SPLINE
SPL {X  -162.820, Y  +617.582, Z    +0.000, E1   +24.552, E3 +451834.871}
SPL {X  -162.820, Y  +614.716, Z    +0.000, E1   +24.535, E3 +451848.082}
SPL {X  -162.820, Y  +611.754, Z    +0.000, E1   +24.563, E3 +451861.370}
SPL {X  -162.820, Y  +608.970, Z    +0.000, E1   +24.542, E3 +451874.211}
SPL {X  -162.820, Y  +606.285, Z    +0.000, E1   +24.533, E3 +451886.546}
SPL {X  -162.820, Y  +603.509, Z    +0.000, E1   +24.546, E3 +451899.084}
SPL {X  -162.820, Y  +600.818, Z    +0.000, E1   +24.590, E3 +451911.006}
SPL {X  -162.820, Y  +598.053, Z    +0.000, E1   +24.547, E3 +451923.989}
SPL {X  -162.820, Y  +595.188, Z    +0.000, E1   +24.538, E3 +451937.078}
SPL {X  -162.820, Y  +592.738, Z    +0.000, E1   +24.551, E3 +451948.126}
SPL {X  -162.820, Y  +590.118, Z    +0.000, E1   +24.544, E3 +451960.185}
SPL {X  -162.820, Y  +587.204, Z    +0.000, E1   +24.592, E3 +451973.062}
SPL {X  -162.820, Y  +584.766, Z    +0.000, E1   +24.499, E3 +451984.895}
SPL {X  -162.820, Y  +581.896, Z    +0.000, E1   +24.528, E3 +451997.837}
SPL {X  -162.820, Y  +579.244, Z    +0.000, E1   +24.610, E3 +452009.181}
SPL {X  -162.820, Y  +576.848, Z    +0.000, E1   +24.543, E3 +452020.723}
SPL {X  -162.820, Y  +574.433, Z    +0.000, E1   +24.551, E3 +452031.553}
SPL {X  -162.820, Y  +572.074, Z    +0.000, E1   +24.505, E3 +452042.824}
SPL {X  -162.820, Y  +568.309, Z    +0.000, E1   +24.589, E3 +452059.451}
SPL {X  -162.820, Y  +564.977, Z    +0.000, E1   +24.571, E3 +452074.624}
SPL {X  -162.820, Y  +562.356, Z    +0.000, E1   +24.575, E3 +452086.523}
SPL {X  -162.820, Y  +558.990, Z    +0.000, E1   +24.558, E3 +452102.173}
SPL {X  -162.820, Y  +555.584, Z    +0.000, E1   +24.559, E3 +452117.541}
SPL {X  -162.820, Y  +552.867, Z    +0.000, E1   +24.583, E3 +452129.737}
SPL {X  -162.820, Y  +549.589, Z    +0.000, E1   +24.547, E3 +452145.103}
SPL {X  -162.820, Y  +545.742, Z    +0.000, E1   +24.577, E3 +452162.390}
SPL {X  -162.820, Y  +542.142, Z    +0.000, E1   +24.582, E3 +452178.743}
SPL {X  -162.820, Y  +538.903, Z    +0.000, E1   +24.519, E3 +452193.959}
SPL {X  -162.820, Y  +536.451, Z    +0.000, E1   +24.519, E3 +452205.039}
SPL {X  -162.820, Y  +534.025, Z    +0.000, E1   +24.589, E3 +452215.639}
SPL {X  -162.820, Y  +531.527, Z    +0.000, E1   +24.582, E3 +452227.024}
SPL {X  -162.820, Y  +529.165, Z    +0.000, E1   +24.521, E3 +452238.273}
SPL {X  -162.820, Y  +525.802, Z    +0.000, E1   +24.585, E3 +452253.293}
SPL {X  -162.820, Y  +521.731, Z    +0.000, E1   +24.542, E3 +452272.229}
SPL {X  -162.820, Y  +518.185, Z    +0.000, E1   +24.561, E3 +452288.101}
SPL {X  -162.820, Y  +508.728, Z    +0.000, E1   +28.484, E3 +452298.641}
SPL {X  -162.820, Y  +500.664, Z    +0.000, E1   +31.476, E3 +452307.305}
SPL {X  -162.820, Y  +499.290, Z    +0.000, E1   +30.657, E3 +452317.587}
SPL {X  -162.820, Y  +497.251, Z    +0.000, E1   +29.634, E3 +452332.063}
SPL {X  -162.820, Y  +495.647, Z    +0.000, E1   +28.606, E3 +452344.939}
SPL {X  -162.820, Y  +494.678, Z    +0.000, E1   +27.647, E3 +452355.640}
SPL {X  -162.820, Y  +493.757, Z    +0.000, E1   +26.462, E3 +452368.000}
SPL {X  -162.820, Y  +492.330, Z    +0.000, E1   +25.953, E3 +452377.754}
SPL {X  -162.820, Y  +489.800, Z    +0.000, E1   +25.653, E3 +452391.216}
SPL {X  -162.820, Y  +485.392, Z    +0.000, E1   +25.667, E3 +452410.243}
SPL {X  -162.820, Y  +482.092, Z    +0.000, E1   +25.593, E3 +452424.931}
SPL {X  -162.820, Y  +479.578, Z    +0.000, E1   +25.634, E3 +452435.574}
SPL {X  -162.820, Y  +476.226, Z    +0.000, E1   +25.672, E3 +452449.964}
SPL {X  -162.820, Y  +473.037, Z    +0.000, E1   +25.618, E3 +452464.055}
SPL {X  -162.820, Y  +469.694, Z    +0.000, E1   +25.657, E3 +452478.430}
SPL {X  -162.820, Y  +465.727, Z    +0.000, E1   +25.676, E3 +452495.473}
SPL {X  -162.820, Y  +463.001, Z    +0.000, E1   +25.614, E3 +452507.589}
SPL {X  -162.820, Y  +459.882, Z    +0.000, E1   +25.674, E3 +452520.890}
SPL {X  -162.820, Y  +456.773, Z    +0.000, E1   +25.591, E3 +452534.836}
SPL {X  -162.820, Y  +454.429, Z    +0.000, E1   +25.642, E3 +452544.604}
SPL {X  -162.820, Y  +451.204, Z    +0.000, E1   +25.672, E3 +452558.631}
SPL {X  -162.820, Y  +447.822, Z    +0.000, E1   +25.664, E3 +452573.114}
SPL {X  -162.820, Y  +445.556, Z    +0.000, E1   +25.626, E3 +452583.245}
SPL {X  -162.820, Y  +443.328, Z    +0.000, E1   +25.642, E3 +452592.759}
SPL {X  -162.820, Y  +440.857, Z    +0.000, E1   +25.614, E3 +452603.794}
SPL {X  -162.820, Y  +437.636, Z    +0.000, E1   +25.597, E3 +452617.957}
SPL {X  -162.820, Y  +434.768, Z    +0.000, E1   +25.655, E3 +452629.859}
SPL {X  -162.820, Y  +431.823, Z    +0.000, E1   +25.651, E3 +452642.858}
SPL {X  -162.820, Y  +427.740, Z    +0.000, E1   +25.667, E3 +452660.486}
SPL {X  -162.820, Y  +423.655, Z    +0.000, E1   +25.628, E3 +452678.510}
SPL {X  -162.820, Y  +419.407, Z    +0.000, E1   +25.665, E3 +452696.703}
SPL {X  -162.820, Y  +415.900, Z    +0.000, E1   +25.638, E3 +452711.972}
SPL {X  -162.820, Y  +413.088, Z    +0.000, E1   +25.644, E3 +452724.128}
SPL {X  -162.820, Y  +410.320, Z    +0.000, E1   +25.604, E3 +452736.447}
SPL {X  -162.820, Y  +407.487, Z    +0.000, E1   +25.617, E3 +452748.655}
SPL {X  -162.820, Y  +404.293, Z    +0.000, E1   +25.628, E3 +452762.564}
SPL {X  -162.820, Y  +400.835, Z    +0.000, E1   +25.694, E3 +452776.964}
SPL {X  -162.820, Y  +398.703, Z    +0.000, E1   +25.586, E3 +452786.956}
SPL {X  -162.820, Y  +396.431, Z    +0.000, E1   +25.636, E3 +452796.479}
SPL {X  -162.820, Y  +393.659, Z    +0.000, E1   +25.666, E3 +452808.329}
SPL {X  -162.820, Y  +390.679, Z    +0.000, E1   +25.624, E3 +452821.573}
SPL {X  -162.820, Y  +387.939, Z    +0.000, E1   +25.627, E3 +452833.432}
SPL {X  -162.820, Y  +384.398, Z    +0.000, E1   +25.707, E3 +452848.330}
SPL {X  -162.820, Y  +380.448, Z    +0.000, E1   +25.674, E3 +452865.694}
SPL {X  -162.785, Y  +377.106, Z    +0.000, E1   +25.598, E3 +452880.638}
SPL {X  -162.709, Y  +374.484, Z    +0.000, E1   +25.711, E3 +452891.089}
SPL {X  -162.623, Y  +372.485, Z    +0.000, E1   +25.631, E3 +452900.369}
SPL {X  -162.487, Y  +370.088, Z    +0.000, E1   +25.525, E3 +452911.623}
SPL {X  -162.243, Y  +366.801, Z    +0.000, E1   +25.618, E3 +452925.264}
SPL {X  -161.882, Y  +363.046, Z    +0.000, E1   +25.550, E3 +452942.147}
SPL {X  -161.454, Y  +359.455, Z    +0.000, E1   +25.428, E3 +452958.541}
SPL {X  -160.939, Y  +355.820, Z    +0.000, E1   +26.179, E3 +452968.424}
SPL {X  -154.424, Y  +328.890, Z    +0.000, E1   +36.591, E3 +452989.256}
ENDSPLINE

SPLINE
SPL {X  -159.701, Y  +348.785, Z    +0.000, E1   +24.361, E3 +453017.539}
SPL {X  -161.904, Y  +363.251, Z    +0.000, E1   +14.606, E3 +453047.335}
SPL {X  -162.745, Y  +375.561, Z    +0.000, E1    +7.538, E3 +453047.531}
SPL {X  -162.820, Y  +385.424, Z    +0.000, E1    +1.080, E3 +453048.425}
SPL {X  -162.820, Y  +389.940, Z    +0.000, E1    -2.281, E3 +453051.302}
SPL {X  -162.820, Y  +396.652, Z    +0.000, E1    -7.520, E3 +453050.881}
SPL {X  -162.820, Y  +406.605, Z    +0.000, E1   -16.760, E3 +453043.357}
SPL {X  -162.820, Y  +418.675, Z    +0.000, E1   -22.201, E3 +453069.606}
SPL {X  -162.820, Y  +425.113, Z    +0.000, E1   -25.243, E3 +453078.542}
SPL {X  -162.820, Y  +441.937, Z    +0.000, E1   -31.578, E3 +453100.620}
ENDSPLINE

SPLINE
SPL {X  -162.820, Y  +437.771, Z    +0.000, E1   -26.555, E3 +453119.721}
ENDSPLINE

SPLINE
SPL {X  -162.820, Y  +439.120, Z    +0.000, E1   -25.352, E3 +453134.264}
SPL {X  -162.820, Y  +441.593, Z    +0.000, E1   -25.391, E3 +453144.816}
SPL {X  -162.820, Y  +444.317, Z    +0.000, E1   -25.492, E3 +453155.997}
SPL {X  -162.820, Y  +446.544, Z    +0.000, E1   -25.427, E3 +453166.167}
SPL {X  -162.820, Y  +448.500, Z    +0.000, E1   -25.425, E3 +453174.768}
SPL {X  -162.820, Y  +451.056, Z    +0.000, E1   -25.443, E3 +453185.876}
SPL {X  -162.820, Y  +454.662, Z    +0.000, E1   -25.474, E3 +453201.620}
SPL {X  -162.820, Y  +458.079, Z    +0.000, E1   -25.369, E3 +453217.199}
SPL {X  -162.820, Y  +460.719, Z    +0.000, E1   -25.411, E3 +453228.457}
SPL {X  -162.820, Y  +463.419, Z    +0.000, E1   -25.510, E3 +453239.495}
SPL {X  -162.820, Y  +465.376, Z    +0.000, E1   -25.372, E3 +453249.083}
SPL {X  -162.820, Y  +467.440, Z    +0.000, E1   -25.427, E3 +453257.714}
SPL {X  -162.820, Y  +470.010, Z    +0.000, E1   -25.445, E3 +453268.919}
SPL {X  -162.820, Y  +473.445, Z    +0.000, E1   -25.493, E3 +453283.643}
SPL {X  -162.820, Y  +476.157, Z    +0.000, E1   -25.426, E3 +453295.858}
SPL {X  -162.820, Y  +478.461, Z    +0.000, E1   -25.410, E3 +453306.137}
SPL {X  -162.820, Y  +481.644, Z    +0.000, E1   -25.433, E3 +453320.084}
SPL {X  -162.820, Y  +486.042, Z    +0.000, E1   -25.483, E3 +453339.003}
SPL {X  -162.820, Y  +490.287, Z    +0.000, E1   -25.463, E3 +453357.721}
SPL {X  -162.820, Y  +494.454, Z    +0.000, E1   -25.465, E3 +453375.953}
SPL {X  -162.820, Y  +498.644, Z    +0.000, E1   -25.463, E3 +453394.329}
SPL {X  -162.820, Y  +502.003, Z    +0.000, E1   -25.416, E3 +453409.227}
SPL {X  -162.820, Y  +505.370, Z    +0.000, E1   -25.456, E3 +453423.803}
SPL {X  -162.820, Y  +509.412, Z    +0.000, E1   -25.458, E3 +453441.525}
SPL {X  -162.820, Y  +512.406, Z    +0.000, E1   -25.425, E3 +453454.682}
SPL {X  -162.820, Y  +515.039, Z    +0.000, E1   -25.452, E3 +453466.092}
SPL {X  -162.820, Y  +518.350, Z    +0.000, E1   -25.425, E3 +453480.842}
SPL {X  -162.820, Y  +521.486, Z    +0.000, E1   -25.382, E3 +453494.869}
SPL {X  -162.820, Y  +524.180, Z    +0.000, E1   -25.495, E3 +453505.742}
SPL {X  -162.820, Y  +527.020, Z    +0.000, E1   -25.477, E3 +453518.434}
SPL {X  -162.820, Y  +529.670, Z    +0.000, E1   -25.472, E3 +453529.892}
SPL {X  -162.820, Y  +532.006, Z    +0.000, E1   -25.455, E3 +453540.349}
SPL {X  -162.820, Y  +534.806, Z    +0.000, E1   -25.465, E3 +453552.465}
SPL {X  -162.820, Y  +537.226, Z    +0.000, E1   -25.378, E3 +453563.747}
SPL {X  -162.820, Y  +540.345, Z    +0.000, E1   -25.451, E3 +453576.928}
SPL {X  -162.820, Y  +543.279, Z    +0.000, E1   -25.419, E3 +453589.961}
SPL {X  -162.820, Y  +546.125, Z    +0.000, E1   -25.505, E3 +453601.755}
SPL {X  -162.820, Y  +549.578, Z    +0.000, E1   -25.462, E3 +453617.379}
SPL {X  -162.820, Y  +553.157, Z    +0.000, E1   -25.443, E3 +453633.043}
SPL {X  -162.820, Y  +556.150, Z    +0.000, E1   -25.445, E3 +453646.133}
SPL {X  -162.820, Y  +559.215, Z    +0.000, E1   -25.460, E3 +453659.434}
SPL {X  -162.820, Y  +562.125, Z    +0.000, E1   -25.434, E3 +453672.355}
SPL {X  -162.820, Y  +565.606, Z    +0.000, E1   -25.468, E3 +453687.484}
SPL {X  -162.820, Y  +568.974, Z    +0.000, E1   -25.453, E3 +453702.195}
SPL {X  -162.820, Y  +571.303, Z    +0.000, E1   -25.427, E3 +453712.541}
SPL {X  -162.820, Y  +574.067, Z    +0.000, E1   -25.459, E3 +453724.480}
SPL {X  -162.820, Y  +576.597, Z    +0.000, E1   -25.400, E3 +453735.951}
SPL {X  -162.820, Y  +580.038, Z    +0.000, E1   -25.473, E3 +453750.647}
SPL {X  -162.820, Y  +583.044, Z    +0.000, E1   -25.450, E3 +453763.770}
SPL {X  -162.820, Y  +585.512, Z    +0.000, E1   -25.448, E3 +453774.665}
SPL {X  -162.820, Y  +588.371, Z    +0.000, E1   -25.460, E3 +453787.051}
SPL {X  -162.820, Y  +590.476, Z    +0.000, E1   -25.398, E3 +453796.693}
SPL {X  -162.820, Y  +593.604, Z    +0.000, E1   -25.477, E3 +453809.971}
SPL {X  -162.820, Y  +596.868, Z    +0.000, E1   -25.461, E3 +453824.236}
SPL {X  -162.820, Y  +599.135, Z    +0.000, E1   -25.398, E3 +453834.605}
SPL {X  -162.820, Y  +601.296, Z    +0.000, E1   -25.399, E3 +453844.087}
SPL {X  -162.820, Y  +604.526, Z    +0.000, E1   -25.502, E3 +453857.581}
SPL {X  -162.820, Y  +607.811, Z    +0.000, E1   -25.507, E3 +453871.795}
SPL {X  -162.820, Y  +610.517, Z    +0.000, E1   -25.412, E3 +453884.358}
SPL {X  -162.820, Y  +613.762, Z    +0.000, E1   -25.472, E3 +453898.165}
SPL {X  -162.820, Y  +617.275, Z    +0.000, E1   -25.466, E3 +453913.603}
SPL {X  -162.820, Y  +619.899, Z    +0.000, E1   -25.455, E3 +453925.008}
SPL {X  -162.820, Y  +622.118, Z    +0.000, E1   -25.492, E3 +453934.475}
SPL {X  -162.820, Y  +624.430, Z    +0.000, E1   -25.475, E3 +453944.696}
SPL {X  -162.820, Y  +626.570, Z    +0.000, E1   -25.441, E3 +453954.296}
SPL {X  -162.820, Y  +628.902, Z    +0.000, E1   -25.449, E3 +453964.476}
SPL {X  -162.820, Y  +631.177, Z    +0.000, E1   -25.467, E3 +453974.308}
SPL {X  -162.820, Y  +633.994, Z    +0.000, E1   -25.503, E3 +453986.354}
SPL {X  -162.820, Y  +637.619, Z    +0.000, E1   -25.497, E3 +454002.414}
SPL {X  -162.820, Y  +640.803, Z    +0.000, E1   -25.462, E3 +454016.377}
SPL {X  -162.820, Y  +643.028, Z    +0.000, E1   -25.494, E3 +454025.886}
SPL {X  -162.820, Y  +646.519, Z    +0.000, E1   -25.551, E3 +454040.868}
SPL {X  -162.820, Y  +649.837, Z    +0.000, E1   -25.446, E3 +454055.993}
SPL {X  -162.820, Y  +652.810, Z    +0.000, E1   -25.497, E3 +454068.635}
SPL {X  -162.820, Y  +655.214, Z    +0.000, E1   -25.485, E3 +454079.138}
SPL {X  -162.820, Y  +657.616, Z    +0.000, E1   -25.511, E3 +454089.492}
SPL {X  -162.820, Y  +660.851, Z    +0.000, E1   -25.520, E3 +454103.635}
SPL {X  -162.820, Y  +663.853, Z    +0.000, E1   -25.496, E3 +454116.816}
SPL {X  -162.820, Y  +667.253, Z    +0.000, E1   -25.483, E3 +454131.989}
SPL {X  -162.820, Y  +671.102, Z    +0.000, E1   -25.514, E3 +454148.439}
SPL {X  -162.820, Y  +673.648, Z    +0.000, E1   -25.431, E3 +454160.106}
SPL {X  -162.796, Y  +676.319, Z    +0.000, E1   -25.526, E3 +454171.116}
SPL {X  -162.707, Y  +679.552, Z    +0.000, E1   -25.443, E3 +454185.990}
SPL {X  -162.545, Y  +682.952, Z    +0.000, E1   -25.510, E3 +454200.223}
SPL {X  -162.381, Y  +685.455, Z    +0.000, E1   -25.410, E3 +454211.910}
SPL {X  -162.102, Y  +688.774, Z    +0.000, E1   -25.417, E3 +454226.524}
SPL {X  -161.711, Y  +692.468, Z    +0.000, E1   -25.300, E3 +454243.497}
SPL {X  -160.732, Y  +699.494, Z    +0.000, E1   -27.462, E3 +454256.969}
SPL {X  -157.189, Y  +715.948, Z    +0.000, E1   -34.218, E3 +454269.127}
ENDSPLINE

SPLINE
SPL {X  -160.780, Y  +699.193, Z    +0.000, E1   -22.069, E3 +454301.039}
ENDSPLINE

SPLINE
SPL {X  -160.671, Y  +699.864, Z    +0.000, E1   -21.788, E3 +454308.470}
ENDSPLINE

SPLINE
SPL {X  -160.945, Y  +698.140, Z    +0.000, E1   -18.412, E3 +454346.038}
SPL {X  -162.497, Y  +683.755, Z    +0.000, E1   -10.754, E3 +454340.182}
SPL {X  -162.819, Y  +673.996, Z    +0.000, E1    -4.745, E3 +454339.783}
ENDSPLINE

SPLINE
SPL {X  -162.791, Y  +676.574, Z    +0.000, E1    -6.127, E3 +454352.471}
ENDSPLINE

SPLINE
SPL {X  -162.820, Y  +666.063, Z    +0.000, E1    +0.780, E3 +454340.564}
SPL {X  -162.820, Y  +659.251, Z    +0.000, E1    +5.716, E3 +454346.781}
SPL {X  -162.820, Y  +640.102, Z    +0.000, E1   +22.409, E3 +454342.560}
SPL {X  -162.820, Y  +633.503, Z    +0.000, E1   +21.975, E3 +454374.796}
SPL {X  -162.820, Y  +611.299, Z    +0.000, E1   +31.088, E3 +454402.909}
ENDSPLINE

SPLINE
SPL {X  -162.820, Y  +618.877, Z    +0.000, E1   +25.259, E3 +454414.403}
ENDSPLINE

SPLINE
SPL {X  -162.820, Y  +617.582, Z    +0.000, E1   +24.552, E3 +454425.780}
SPL {X  -162.820, Y  +614.716, Z    +0.000, E1   +24.535, E3 +454438.991}
SPL {X  -162.820, Y  +611.754, Z    +0.000, E1   +24.563, E3 +454452.280}
SPL {X  -162.820, Y  +608.970, Z    +0.000, E1   +24.542, E3 +454465.120}
SPL {X  -162.820, Y  +606.285, Z    +0.000, E1   +24.533, E3 +454477.455}
SPL {X  -162.820, Y  +603.509, Z    +0.000, E1   +24.546, E3 +454489.993}
SPL {X  -162.820, Y  +600.818, Z    +0.000, E1   +24.590, E3 +454501.915}
SPL {X  -162.820, Y  +598.053, Z    +0.000, E1   +24.547, E3 +454514.898}
SPL {X  -162.820, Y  +595.188, Z    +0.000, E1   +24.538, E3 +454527.987}
SPL {X  -162.820, Y  +592.738, Z    +0.000, E1   +24.551, E3 +454539.035}
SPL {X  -162.820, Y  +590.118, Z    +0.000, E1   +24.544, E3 +454551.094}
SPL {X  -162.820, Y  +587.204, Z    +0.000, E1   +24.592, E3 +454563.971}
SPL {X  -162.820, Y  +584.766, Z    +0.000, E1   +24.499, E3 +454575.804}
SPL {X  -162.820, Y  +581.896, Z    +0.000, E1   +24.528, E3 +454588.746}
SPL {X  -162.820, Y  +579.244, Z    +0.000, E1   +24.610, E3 +454600.090}
SPL {X  -162.820, Y  +576.848, Z    +0.000, E1   +24.543, E3 +454611.632}
SPL {X  -162.820, Y  +574.433, Z    +0.000, E1   +24.551, E3 +454622.462}
SPL {X  -162.820, Y  +572.074, Z    +0.000, E1   +24.505, E3 +454633.734}
SPL {X  -162.820, Y  +568.309, Z    +0.000, E1   +24.589, E3 +454650.360}
SPL {X  -162.820, Y  +564.977, Z    +0.000, E1   +24.571, E3 +454665.533}
SPL {X  -162.820, Y  +562.356, Z    +0.000, E1   +24.575, E3 +454677.432}
SPL {X  -162.820, Y  +558.990, Z    +0.000, E1   +24.558, E3 +454693.082}
SPL {X  -162.820, Y  +555.584, Z    +0.000, E1   +24.559, E3 +454708.451}
SPL {X  -162.820, Y  +552.169, Z    +0.000, E1   +24.581, E3 +454724.019}
SPL {X  -162.820, Y  +548.172, Z    +0.000, E1   +24.564, E3 +454742.367}
SPL {X  -162.820, Y  +544.025, Z    +0.000, E1   +24.611, E3 +454760.921}
SPL {X  -162.820, Y  +540.573, Z    +0.000, E1   +24.503, E3 +454777.376}
SPL {X  -162.820, Y  +537.211, Z    +0.000, E1   +24.561, E3 +454792.305}
SPL {X  -162.820, Y  +534.025, Z    +0.000, E1   +24.589, E3 +454806.548}
SPL {X  -162.820, Y  +531.527, Z    +0.000, E1   +24.582, E3 +454817.933}
SPL {X  -162.820, Y  +529.165, Z    +0.000, E1   +24.521, E3 +454829.182}
SPL {X  -162.820, Y  +526.822, Z    +0.000, E1   +24.559, E3 +454839.545}
SPL {X  -162.820, Y  +524.112, Z    +0.000, E1   +24.542, E3 +454852.163}
SPL {X  -162.820, Y  +521.048, Z    +0.000, E1   +24.515, E3 +454866.299}
SPL {X  -162.820, Y  +518.185, Z    +0.000, E1   +24.561, E3 +454879.010}
SPL {X  -162.820, Y  +508.728, Z    +0.000, E1   +28.484, E3 +454889.550}
SPL {X  -162.820, Y  +500.664, Z    +0.000, E1   +31.476, E3 +454898.214}
SPL {X  -162.820, Y  +499.290, Z    +0.000, E1   +30.657, E3 +454908.496}
SPL {X  -162.820, Y  +497.700, Z    +0.000, E1   +29.785, E3 +454920.111}
SPL {X  -162.820, Y  +495.915, Z    +0.000, E1   +28.861, E3 +454933.204}
SPL {X  -162.820, Y  +494.678, Z    +0.000, E1   +27.647, E3 +454946.549}
SPL {X  -162.820, Y  +493.757, Z    +0.000, E1   +26.462, E3 +454958.909}
SPL {X  -162.820, Y  +491.420, Z    +0.000, E1   +25.780, E3 +454974.171}
SPL {X  -162.820, Y  +487.351, Z    +0.000, E1   +25.663, E3 +454992.687}
SPL {X  -162.820, Y  +484.247, Z    +0.000, E1   +25.651, E3 +455006.013}
SPL {X  -162.820, Y  +482.092, Z    +0.000, E1   +25.593, E3 +455015.840}
SPL {X  -162.820, Y  +479.578, Z    +0.000, E1   +25.634, E3 +455026.483}
SPL {X  -162.820, Y  +477.137, Z    +0.000, E1   +25.632, E3 +455037.062}
SPL {X  -162.820, Y  +473.770, Z    +0.000, E1   +25.664, E3 +455051.608}
SPL {X  -162.820, Y  +469.694, Z    +0.000, E1   +25.657, E3 +455069.339}
SPL {X  -162.820, Y  +465.727, Z    +0.000, E1   +25.676, E3 +455086.382}
SPL {X  -162.820, Y  +463.001, Z    +0.000, E1   +25.614, E3 +455098.498}
SPL {X  -162.820, Y  +459.882, Z    +0.000, E1   +25.674, E3 +455111.799}
SPL {X  -162.820, Y  +456.773, Z    +0.000, E1   +25.591, E3 +455125.745}
SPL {X  -162.820, Y  +454.429, Z    +0.000, E1   +25.642, E3 +455135.513}
SPL {X  -162.820, Y  +451.204, Z    +0.000, E1   +25.672, E3 +455149.540}
SPL {X  -162.820, Y  +447.822, Z    +0.000, E1   +25.664, E3 +455164.023}
SPL {X  -162.820, Y  +445.556, Z    +0.000, E1   +25.626, E3 +455174.154}
SPL {X  -162.820, Y  +442.508, Z    +0.000, E1   +25.657, E3 +455187.248}
SPL {X  -162.820, Y  +439.273, Z    +0.000, E1   +25.576, E3 +455201.886}
SPL {X  -162.820, Y  +436.773, Z    +0.000, E1   +25.602, E3 +455212.451}
SPL {X  -162.820, Y  +433.761, Z    +0.000, E1   +25.681, E3 +455225.129}
SPL {X  -162.820, Y  +430.942, Z    +0.000, E1   +25.597, E3 +455237.814}
SPL {X  -162.820, Y  +428.576, Z    +0.000, E1   +25.647, E3 +455247.752}
SPL {X  -162.820, Y  +426.525, Z    +0.000, E1   +25.610, E3 +455256.860}
SPL {X  -162.820, Y  +423.655, Z    +0.000, E1   +25.628, E3 +455269.419}
SPL {X  -162.820, Y  +419.407, Z    +0.000, E1   +25.665, E3 +455287.612}
SPL {X  -162.820, Y  +415.900, Z    +0.000, E1   +25.638, E3 +455302.881}
SPL {X  -162.820, Y  +413.088, Z    +0.000, E1   +25.644, E3 +455315.037}
SPL {X  -162.820, Y  +410.320, Z    +0.000, E1   +25.604, E3 +455327.356}
SPL {X  -162.820, Y  +407.487, Z    +0.000, E1   +25.617, E3 +455339.564}
SPL {X  -162.820, Y  +405.108, Z    +0.000, E1   +25.535, E3 +455350.532}
SPL {X  -162.820, Y  +401.373, Z    +0.000, E1   +25.736, E3 +455365.368}
SPL {X  -162.820, Y  +398.703, Z    +0.000, E1   +25.586, E3 +455377.865}
SPL {X  -162.820, Y  +395.582, Z    +0.000, E1   +25.684, E3 +455390.857}
SPL {X  -162.820, Y  +391.417, Z    +0.000, E1   +25.659, E3 +455409.194}
SPL {X  -162.820, Y  +387.939, Z    +0.000, E1   +25.627, E3 +455424.341}
SPL {X  -162.820, Y  +385.565, Z    +0.000, E1   +25.686, E3 +455434.130}
SPL {X  -162.820, Y  +383.458, Z    +0.000, E1   +25.657, E3 +455443.494}
SPL {X  -162.820, Y  +381.229, Z    +0.000, E1   +25.660, E3 +455453.169}
SPL {X  -162.797, Y  +377.786, Z    +0.000, E1   +25.638, E3 +455468.459}
SPL {X  -162.663, Y  +373.346, Z    +0.000, E1   +25.707, E3 +455487.198}
SPL {X  -162.487, Y  +370.088, Z    +0.000, E1   +25.525, E3 +455502.532}
SPL {X  -162.307, Y  +367.587, Z    +0.000, E1   +25.577, E3 +455512.951}
SPL {X  -162.041, Y  +364.588, Z    +0.000, E1   +25.591, E3 +455526.028}
SPL {X  -161.695, Y  +361.389, Z    +0.000, E1   +25.445, E3 +455540.915}
SPL {X  -161.190, Y  +357.520, Z    +0.000, E1   +25.774, E3 +455555.166}
SPL {X  -155.035, Y  +330.756, Z    +0.000, E1   +37.918, E3 +455565.667}
SPL {X  -153.918, Y  +327.401, Z    +0.000, E1   +34.677, E3 +455600.968}
ENDSPLINE

SPLINE
SPL {X  -159.701, Y  +348.785, Z    +0.000, E1   +24.361, E3 +455608.449}
SPL {X  -161.904, Y  +363.251, Z    +0.000, E1   +14.606, E3 +455638.244}
SPL {X  -162.745, Y  +375.561, Z    +0.000, E1    +7.538, E3 +455638.440}
SPL {X  -162.820, Y  +385.424, Z    +0.000, E1    +1.080, E3 +455639.335}
SPL {X  -162.820, Y  +389.940, Z    +0.000, E1    -2.281, E3 +455642.211}
SPL {X  -162.820, Y  +396.652, Z    +0.000, E1    -7.520, E3 +455641.790}
SPL {X  -162.820, Y  +406.605, Z    +0.000, E1   -16.760, E3 +455634.267}
SPL {X  -162.820, Y  +420.013, Z    +0.000, E1   -22.833, E3 +455662.387}
SPL {X  -162.820, Y  +442.075, Z    +0.000, E1   -31.090, E3 +455695.173}
ENDSPLINE

SPLINE
SPL {X  -162.820, Y  +436.680, Z    +0.000, E1   -26.151, E3 +455708.478}
ENDSPLINE

SPLINE
SPL {X  -162.820, Y  +438.487, Z    +0.000, E1   -25.409, E3 +455722.117}
SPL {X  -162.820, Y  +441.593, Z    +0.000, E1   -25.391, E3 +455735.725}
SPL {X  -162.820, Y  +444.317, Z    +0.000, E1   -25.492, E3 +455746.906}
SPL {X  -162.820, Y  +447.641, Z    +0.000, E1   -25.460, E3 +455761.841}
SPL {X  -162.820, Y  +451.939, Z    +0.000, E1   -25.468, E3 +455780.662}
SPL {X  -162.820, Y  +455.480, Z    +0.000, E1   -25.454, E3 +455796.073}
SPL {X  -162.820, Y  +458.079, Z    +0.000, E1   -25.369, E3 +455808.108}
SPL {X  -162.820, Y  +460.719, Z    +0.000, E1   -25.411, E3 +455819.366}
SPL {X  -162.820, Y  +463.419, Z    +0.000, E1   -25.510, E3 +455830.404}
SPL {X  -162.820, Y  +466.458, Z    +0.000, E1   -25.433, E3 +455844.460}
SPL {X  -162.820, Y  +470.010, Z    +0.000, E1   -25.445, E3 +455859.828}
SPL {X  -162.820, Y  +472.345, Z    +0.000, E1   -25.448, E3 +455869.915}
SPL {X  -162.820, Y  +475.191, Z    +0.000, E1   -25.489, E3 +455882.277}
SPL {X  -162.820, Y  +478.461, Z    +0.000, E1   -25.410, E3 +455897.046}
SPL {X  -162.820, Y  +480.780, Z    +0.000, E1   -25.447, E3 +455906.908}
SPL {X  -162.820, Y  +483.622, Z    +0.000, E1   -25.381, E3 +455919.950}
SPL {X  -162.820, Y  +487.570, Z    +0.000, E1   -25.482, E3 +455936.588}
SPL {X  -162.820, Y  +491.017, Z    +0.000, E1   -25.445, E3 +455951.803}
SPL {X  -162.820, Y  +493.705, Z    +0.000, E1   -25.443, E3 +455963.587}
SPL {X  -162.820, Y  +497.247, Z    +0.000, E1   -25.470, E3 +455979.049}
SPL {X  -162.820, Y  +501.343, Z    +0.000, E1   -25.435, E3 +455997.248}
SPL {X  -162.820, Y  +505.370, Z    +0.000, E1   -25.456, E3 +456014.712}
SPL {X  -162.820, Y  +509.412, Z    +0.000, E1   -25.458, E3 +456032.434}
SPL {X  -162.820, Y  +512.406, Z    +0.000, E1   -25.425, E3 +456045.591}
SPL {X  -162.820, Y  +515.039, Z    +0.000, E1   -25.452, E3 +456057.001}
SPL {X  -162.820, Y  +518.350, Z    +0.000, E1   -25.425, E3 +456071.751}
SPL {X  -162.820, Y  +521.486, Z    +0.000, E1   -25.382, E3 +456085.778}
SPL {X  -162.820, Y  +524.180, Z    +0.000, E1   -25.495, E3 +456096.651}
SPL {X  -162.820, Y  +527.020, Z    +0.000, E1   -25.477, E3 +456109.343}
SPL {X  -162.820, Y  +529.670, Z    +0.000, E1   -25.472, E3 +456120.801}
SPL {X  -162.820, Y  +532.006, Z    +0.000, E1   -25.455, E3 +456131.258}
SPL {X  -162.820, Y  +534.806, Z    +0.000, E1   -25.465, E3 +456143.374}
SPL {X  -162.820, Y  +537.226, Z    +0.000, E1   -25.378, E3 +456154.656}
SPL {X  -162.820, Y  +540.345, Z    +0.000, E1   -25.451, E3 +456167.837}
SPL {X  -162.820, Y  +543.279, Z    +0.000, E1   -25.419, E3 +456180.870}
SPL {X  -162.820, Y  +546.125, Z    +0.000, E1   -25.505, E3 +456192.664}
SPL {X  -162.820, Y  +549.578, Z    +0.000, E1   -25.462, E3 +456208.289}
SPL {X  -162.820, Y  +553.157, Z    +0.000, E1   -25.443, E3 +456223.952}
SPL {X  -162.820, Y  +556.150, Z    +0.000, E1   -25.445, E3 +456237.042}
SPL {X  -162.820, Y  +559.215, Z    +0.000, E1   -25.460, E3 +456250.343}
SPL {X  -162.820, Y  +562.125, Z    +0.000, E1   -25.434, E3 +456263.264}
SPL {X  -162.820, Y  +565.606, Z    +0.000, E1   -25.468, E3 +456278.393}
SPL {X  -162.820, Y  +568.974, Z    +0.000, E1   -25.453, E3 +456293.104}
SPL {X  -162.820, Y  +571.303, Z    +0.000, E1   -25.427, E3 +456303.450}
SPL {X  -162.820, Y  +574.067, Z    +0.000, E1   -25.459, E3 +456315.389}
SPL {X  -162.820, Y  +576.597, Z    +0.000, E1   -25.400, E3 +456326.860}
SPL {X  -162.820, Y  +580.038, Z    +0.000, E1   -25.473, E3 +456341.556}
SPL {X  -162.820, Y  +583.044, Z    +0.000, E1   -25.450, E3 +456354.679}
SPL {X  -162.820, Y  +585.512, Z    +0.000, E1   -25.448, E3 +456365.575}
SPL {X  -162.820, Y  +588.371, Z    +0.000, E1   -25.460, E3 +456377.961}
SPL {X  -162.820, Y  +591.246, Z    +0.000, E1   -25.415, E3 +456390.980}
SPL {X  -162.820, Y  +594.339, Z    +0.000, E1   -25.487, E3 +456403.882}
SPL {X  -162.820, Y  +596.868, Z    +0.000, E1   -25.461, E3 +456415.145}
SPL {X  -162.820, Y  +600.326, Z    +0.000, E1   -25.438, E3 +456430.667}
SPL {X  -162.820, Y  +603.808, Z    +0.000, E1   -25.554, E3 +456444.784}
SPL {X  -162.820, Y  +607.007, Z    +0.000, E1   -25.491, E3 +456459.475}
SPL {X  -162.820, Y  +611.438, Z    +0.000, E1   -25.467, E3 +456479.065}
SPL {X  -162.820, Y  +615.388, Z    +0.000, E1   -25.455, E3 +456496.324}
SPL {X  -162.820, Y  +618.103, Z    +0.000, E1   -25.456, E3 +456508.071}
SPL {X  -162.820, Y  +621.264, Z    +0.000, E1   -25.514, E3 +456521.674}
SPL {X  -162.820, Y  +624.430, Z    +0.000, E1   -25.475, E3 +456535.605}
SPL {X  -162.820, Y  +626.570, Z    +0.000, E1   -25.441, E3 +456545.205}
SPL {X  -162.820, Y  +628.902, Z    +0.000, E1   -25.449, E3 +456555.385}
SPL {X  -162.820, Y  +631.177, Z    +0.000, E1   -25.467, E3 +456565.217}
SPL {X  -162.820, Y  +633.994, Z    +0.000, E1   -25.503, E3 +456577.263}
SPL {X  -162.820, Y  +637.619, Z    +0.000, E1   -25.497, E3 +456593.323}
SPL {X  -162.820, Y  +640.803, Z    +0.000, E1   -25.462, E3 +456607.286}
SPL {X  -162.820, Y  +643.028, Z    +0.000, E1   -25.494, E3 +456616.795}
SPL {X  -162.820, Y  +646.519, Z    +0.000, E1   -25.551, E3 +456631.777}
SPL {X  -162.820, Y  +649.837, Z    +0.000, E1   -25.446, E3 +456646.902}
SPL {X  -162.820, Y  +652.810, Z    +0.000, E1   -25.497, E3 +456659.544}
SPL {X  -162.820, Y  +655.214, Z    +0.000, E1   -25.485, E3 +456670.047}
SPL {X  -162.820, Y  +657.616, Z    +0.000, E1   -25.511, E3 +456680.401}
SPL {X  -162.820, Y  +660.851, Z    +0.000, E1   -25.520, E3 +456694.544}
SPL {X  -162.820, Y  +663.853, Z    +0.000, E1   -25.496, E3 +456707.726}
SPL {X  -162.820, Y  +667.253, Z    +0.000, E1   -25.483, E3 +456722.898}
SPL {X  -162.820, Y  +671.102, Z    +0.000, E1   -25.514, E3 +456739.348}
SPL {X  -162.820, Y  +673.648, Z    +0.000, E1   -25.431, E3 +456751.015}
SPL {X  -162.796, Y  +676.319, Z    +0.000, E1   -25.526, E3 +456762.025}
SPL {X  -162.739, Y  +678.625, Z    +0.000, E1   -25.423, E3 +456772.816}
SPL {X  -162.669, Y  +680.515, Z    +0.000, E1   -25.398, E3 +456781.270}
SPL {X  -162.545, Y  +682.952, Z    +0.000, E1   -25.510, E3 +456791.132}
SPL {X  -162.381, Y  +685.455, Z    +0.000, E1   -25.410, E3 +456802.819}
SPL {X  -162.194, Y  +687.760, Z    +0.000, E1   -25.360, E3 +456813.255}
SPL {X  -161.987, Y  +689.945, Z    +0.000, E1   -25.406, E3 +456822.407}
SPL {X  -161.711, Y  +692.468, Z    +0.000, E1   -25.300, E3 +456834.406}
SPL {X  -160.732, Y  +699.494, Z    +0.000, E1   -27.462, E3 +456847.878}
SPL {X  -157.189, Y  +715.948, Z    +0.000, E1   -34.218, E3 +456860.036}
ENDSPLINE

SPLINE
SPL {X  -157.848, Y  +713.428, Z    +0.000, E1   -28.857, E3 +456894.175}
SPL {X  -161.035, Y  +697.541, Z    +0.000, E1   -20.899, E3 +456894.694}
SPL {X  -161.689, Y  +692.657, Z    +0.000, E1   -15.656, E3 +456934.777}
SPL {X  -162.807, Y  +675.545, Z    +0.000, E1    -5.787, E3 +456930.277}
ENDSPLINE

SPLINE
SPL {X  -162.791, Y  +676.574, Z    +0.000, E1    -6.127, E3 +456943.380}
ENDSPLINE

SPLINE
SPL {X  -162.820, Y  +664.716, Z    +0.000, E1    +1.705, E3 +456932.254}
SPL {X  -162.820, Y  +658.484, Z    +0.000, E1    +6.336, E3 +456938.730}
SPL {X  -162.820, Y  +640.102, Z    +0.000, E1   +22.409, E3 +456933.469}
SPL {X  -162.820, Y  +633.503, Z    +0.000, E1   +21.975, E3 +456965.705}
SPL {X  -162.820, Y  +611.299, Z    +0.000, E1   +31.088, E3 +456993.818}
ENDSPLINE

SPLINE
SPL {X  -162.820, Y  +618.877, Z    +0.000, E1   +25.259, E3 +457005.312}
ENDSPLINE

SPLINE
SPL {X  -162.820, Y  +617.582, Z    +0.000, E1   +24.552, E3 +457016.689}
SPL {X  -162.820, Y  +614.716, Z    +0.000, E1   +24.535, E3 +457029.900}
SPL {X  -162.820, Y  +611.754, Z    +0.000, E1   +24.563, E3 +457043.189}
SPL {X  -162.820, Y  +608.970, Z    +0.000, E1   +24.542, E3 +457056.029}
SPL {X  -162.820, Y  +606.285, Z    +0.000, E1   +24.533, E3 +457068.364}
SPL {X  -162.820, Y  +603.509, Z    +0.000, E1   +24.546, E3 +457080.902}
SPL {X  -162.820, Y  +600.818, Z    +0.000, E1   +24.590, E3 +457092.824}
SPL {X  -162.820, Y  +598.053, Z    +0.000, E1   +24.547, E3 +457105.807}
SPL {X  -162.820, Y  +595.188, Z    +0.000, E1   +24.538, E3 +457118.896}
SPL {X  -162.820, Y  +592.738, Z    +0.000, E1   +24.551, E3 +457129.944}
SPL {X  -162.820, Y  +590.118, Z    +0.000, E1   +24.544, E3 +457142.003}
SPL {X  -162.820, Y  +587.204, Z    +0.000, E1   +24.592, E3 +457154.880}
SPL {X  -162.820, Y  +584.766, Z    +0.000, E1   +24.499, E3 +457166.713}
SPL {X  -162.820, Y  +581.896, Z    +0.000, E1   +24.528, E3 +457179.655}
SPL {X  -162.820, Y  +578.588, Z    +0.000, E1   +24.598, E3 +457194.207}
SPL {X  -162.820, Y  +576.196, Z    +0.000, E1   +24.519, E3 +457205.590}
SPL {X  -162.820, Y  +573.694, Z    +0.000, E1   +24.535, E3 +457217.010}
SPL {X  -162.820, Y  +570.310, Z    +0.000, E1   +24.556, E3 +457232.327}
SPL {X  -162.820, Y  +567.494, Z    +0.000, E1   +24.547, E3 +457245.112}
SPL {X  -162.820, Y  +564.977, Z    +0.000, E1   +24.571, E3 +457256.442}
SPL {X  -162.820, Y  +562.356, Z    +0.000, E1   +24.575, E3 +457268.341}
SPL {X  -162.820, Y  +558.990, Z    +0.000, E1   +24.558, E3 +457283.991}
SPL {X  -162.820, Y  +555.584, Z    +0.000, E1   +24.559, E3 +457299.360}
SPL {X  -162.820, Y  +552.169, Z    +0.000, E1   +24.581, E3 +457314.929}
SPL {X  -162.820, Y  +548.172, Z    +0.000, E1   +24.564, E3 +457333.276}
SPL {X  -162.820, Y  +544.025, Z    +0.000, E1   +24.611, E3 +457351.831}
SPL {X  -162.820, Y  +540.573, Z    +0.000, E1   +24.503, E3 +457368.285}
SPL {X  -162.820, Y  +538.106, Z    +0.000, E1   +24.553, E3 +457379.039}
SPL {X  -162.820, Y  +536.451, Z    +0.000, E1   +24.519, E3 +457386.857}
SPL {X  -162.820, Y  +534.025, Z    +0.000, E1   +24.589, E3 +457397.457}
SPL {X  -162.820, Y  +531.527, Z    +0.000, E1   +24.582, E3 +457408.843}
SPL {X  -162.820, Y  +529.165, Z    +0.000, E1   +24.521, E3 +457420.091}
SPL {X  -162.820, Y  +526.822, Z    +0.000, E1   +24.559, E3 +457430.455}
SPL {X  -162.820, Y  +524.112, Z    +0.000, E1   +24.542, E3 +457443.072}
SPL {X  -162.820, Y  +521.048, Z    +0.000, E1   +24.515, E3 +457457.209}
SPL {X  -162.820, Y  +518.185, Z    +0.000, E1   +24.561, E3 +457469.920}
SPL {X  -162.820, Y  +508.728, Z    +0.000, E1   +28.484, E3 +457480.459}
SPL {X  -162.820, Y  +500.664, Z    +0.000, E1   +31.476, E3 +457489.123}
SPL {X  -162.820, Y  +499.290, Z    +0.000, E1   +30.657, E3 +457499.405}
SPL {X  -162.820, Y  +497.251, Z    +0.000, E1   +29.634, E3 +457513.881}
SPL {X  -162.820, Y  +495.647, Z    +0.000, E1   +28.606, E3 +457526.757}
SPL {X  -162.820, Y  +494.678, Z    +0.000, E1   +27.647, E3 +457537.458}
SPL {X  -162.820, Y  +493.757, Z    +0.000, E1   +26.462, E3 +457549.818}
SPL {X  -162.820, Y  +492.330, Z    +0.000, E1   +25.953, E3 +457559.572}
SPL {X  -162.820, Y  +489.800, Z    +0.000, E1   +25.653, E3 +457573.034}
SPL {X  -162.820, Y  +485.392, Z    +0.000, E1   +25.667, E3 +457592.061}
SPL {X  -162.820, Y  +482.092, Z    +0.000, E1   +25.593, E3 +457606.749}
SPL {X  -162.820, Y  +479.578, Z    +0.000, E1   +25.634, E3 +457617.392}
SPL {X  -162.820, Y  +476.226, Z    +0.000, E1   +25.672, E3 +457631.783}
SPL {X  -162.820, Y  +473.037, Z    +0.000, E1   +25.618, E3 +457645.873}
SPL {X  -162.820, Y  +470.744, Z    +0.000, E1   +25.641, E3 +457655.614}
SPL {X  -162.820, Y  +467.745, Z    +0.000, E1   +25.668, E3 +457668.596}
SPL {X  -162.820, Y  +463.978, Z    +0.000, E1   +25.651, E3 +457685.074}
SPL {X  -162.820, Y  +459.882, Z    +0.000, E1   +25.674, E3 +457702.708}
SPL {X  -162.820, Y  +456.773, Z    +0.000, E1   +25.591, E3 +457716.654}
SPL {X  -162.820, Y  +454.429, Z    +0.000, E1   +25.642, E3 +457726.422}
SPL {X  -162.820, Y  +451.204, Z    +0.000, E1   +25.672, E3 +457740.449}
SPL {X  -162.820, Y  +447.822, Z    +0.000, E1   +25.664, E3 +457754.933}
SPL {X  -162.820, Y  +445.556, Z    +0.000, E1   +25.626, E3 +457765.063}
SPL {X  -162.820, Y  +442.508, Z    +0.000, E1   +25.657, E3 +457778.157}
SPL {X  -162.820, Y  +439.273, Z    +0.000, E1   +25.576, E3 +457792.795}
SPL {X  -162.820, Y  +436.773, Z    +0.000, E1   +25.602, E3 +457803.360}
SPL {X  -162.820, Y  +433.761, Z    +0.000, E1   +25.681, E3 +457816.038}
SPL {X  -162.820, Y  +430.942, Z    +0.000, E1   +25.597, E3 +457828.724}
SPL {X  -162.820, Y  +428.576, Z    +0.000, E1   +25.647, E3 +457838.661}
SPL {X  -162.820, Y  +425.120, Z    +0.000, E1   +25.647, E3 +457853.845}
SPL {X  -162.820, Y  +420.840, Z    +0.000, E1   +25.658, E3 +457872.352}
SPL {X  -162.820, Y  +416.590, Z    +0.000, E1   +25.659, E3 +457890.796}
SPL {X  -162.820, Y  +412.302, Z    +0.000, E1   +25.662, E3 +457909.402}
SPL {X  -162.820, Y  +408.133, Z    +0.000, E1   +25.637, E3 +457927.660}
SPL {X  -162.820, Y  +404.293, Z    +0.000, E1   +25.628, E3 +457944.382}
SPL {X  -162.820, Y  +400.835, Z    +0.000, E1   +25.694, E3 +457958.782}
SPL {X  -162.820, Y  +398.703, Z    +0.000, E1   +25.586, E3 +457968.774}
SPL {X  -162.820, Y  +395.582, Z    +0.000, E1   +25.684, E3 +457981.766}
SPL {X  -162.820, Y  +391.417, Z    +0.000, E1   +25.659, E3 +458000.104}
SPL {X  -162.820, Y  +387.939, Z    +0.000, E1   +25.627, E3 +458015.250}
SPL {X  -162.820, Y  +385.565, Z    +0.000, E1   +25.686, E3 +458025.039}
SPL {X  -162.820, Y  +383.458, Z    +0.000, E1   +25.657, E3 +458034.403}
SPL {X  -162.820, Y  +381.229, Z    +0.000, E1   +25.660, E3 +458044.078}
SPL {X  -162.797, Y  +377.786, Z    +0.000, E1   +25.638, E3 +458059.368}
SPL {X  -162.663, Y  +373.346, Z    +0.000, E1   +25.707, E3 +458078.107}
SPL {X  -162.487, Y  +370.088, Z    +0.000, E1   +25.525, E3 +458093.442}
SPL {X  -162.307, Y  +367.587, Z    +0.000, E1   +25.577, E3 +458103.860}
SPL {X  -162.041, Y  +364.588, Z    +0.000, E1   +25.591, E3 +458116.938}
SPL {X  -161.695, Y  +361.389, Z    +0.000, E1   +25.445, E3 +458131.824}
SPL {X  -161.364, Y  +358.774, Z    +0.000, E1   +25.454, E3 +458143.024}
SPL {X  -160.939, Y  +355.820, Z    +0.000, E1   +26.179, E3 +458150.242}
SPL {X  -155.035, Y  +330.756, Z    +0.000, E1   +37.918, E3 +458156.576}
SPL {X  -153.918, Y  +327.401, Z    +0.000, E1   +34.677, E3 +458191.877}
ENDSPLINE

SPLINE
SPL {X  -159.701, Y  +348.785, Z    +0.000, E1   +24.361, E3 +458199.358}
SPL {X  -161.904, Y  +363.251, Z    +0.000, E1   +14.606, E3 +458229.153}
SPL {X  -162.745, Y  +375.561, Z    +0.000, E1    +7.538, E3 +458229.349}
SPL {X  -162.820, Y  +385.424, Z    +0.000, E1    +1.080, E3 +458230.244}
SPL {X  -162.820, Y  +389.940, Z    +0.000, E1    -2.281, E3 +458233.120}
SPL {X  -162.820, Y  +396.652, Z    +0.000, E1    -7.520, E3 +458232.699}
SPL {X  -162.820, Y  +406.605, Z    +0.000, E1   -16.760, E3 +458225.176}
SPL {X  -162.820, Y  +420.013, Z    +0.000, E1   -22.833, E3 +458253.296}
SPL {X  -162.820, Y  +442.075, Z    +0.000, E1   -31.090, E3 +458286.083}
ENDSPLINE

SPLINE
SPL {X  -162.820, Y  +436.680, Z    +0.000, E1   -26.151, E3 +458299.387}
ENDSPLINE

SPLINE
SPL {X  -162.820, Y  +438.487, Z    +0.000, E1   -25.409, E3 +458313.026}
SPL {X  -162.820, Y  +441.593, Z    +0.000, E1   -25.391, E3 +458326.634}
SPL {X  -162.820, Y  +444.317, Z    +0.000, E1   -25.492, E3 +458337.815}
SPL {X  -162.820, Y  +446.544, Z    +0.000, E1   -25.427, E3 +458347.985}
SPL {X  -162.820, Y  +448.500, Z    +0.000, E1   -25.425, E3 +458356.586}
SPL {X  -162.820, Y  +451.939, Z    +0.000, E1   -25.468, E3 +458371.571}
SPL {X  -162.820, Y  +455.480, Z    +0.000, E1   -25.454, E3 +458386.982}
SPL {X  -162.820, Y  +458.079, Z    +0.000, E1   -25.369, E3 +458399.017}
SPL {X  -162.820, Y  +460.719, Z    +0.000, E1   -25.411, E3 +458410.275}
SPL {X  -162.820, Y  +463.419, Z    +0.000, E1   -25.510, E3 +458421.313}
SPL {X  -162.820, Y  +466.458, Z    +0.000, E1   -25.433, E3 +458435.369}
SPL {X  -162.820, Y  +470.010, Z    +0.000, E1   -25.445, E3 +458450.737}
SPL {X  -162.820, Y  +472.345, Z    +0.000, E1   -25.448, E3 +458460.824}
SPL {X  -162.820, Y  +475.191, Z    +0.000, E1   -25.489, E3 +458473.186}
SPL {X  -162.820, Y  +478.461, Z    +0.000, E1   -25.410, E3 +458487.955}
SPL {X  -162.820, Y  +480.780, Z    +0.000, E1   -25.447, E3 +458497.817}
SPL {X  -162.820, Y  +483.622, Z    +0.000, E1   -25.381, E3 +458510.859}
SPL {X  -162.820, Y  +487.570, Z    +0.000, E1   -25.482, E3 +458527.497}
SPL {X  -162.820, Y  +491.017, Z    +0.000, E1   -25.445, E3 +458542.712}
SPL {X  -162.820, Y  +494.454, Z    +0.000, E1   -25.465, E3 +458557.771}
SPL {X  -162.820, Y  +498.644, Z    +0.000, E1   -25.463, E3 +458576.147}
SPL {X  -162.820, Y  +502.845, Z    +0.000, E1   -25.458, E3 +458594.580}
SPL {X  -162.820, Y  +506.050, Z    +0.000, E1   -25.420, E3 +458608.720}
SPL {X  -162.820, Y  +508.346, Z    +0.000, E1   -25.444, E3 +458618.568}
SPL {X  -162.820, Y  +511.422, Z    +0.000, E1   -25.445, E3 +458632.229}
SPL {X  -162.820, Y  +515.039, Z    +0.000, E1   -25.452, E3 +458647.910}
SPL {X  -162.820, Y  +518.350, Z    +0.000, E1   -25.425, E3 +458662.660}
SPL {X  -162.820, Y  +521.486, Z    +0.000, E1   -25.382, E3 +458676.687}
SPL {X  -162.820, Y  +524.180, Z    +0.000, E1   -25.495, E3 +458687.560}
SPL {X  -162.820, Y  +527.020, Z    +0.000, E1   -25.477, E3 +458700.253}
SPL {X  -162.820, Y  +529.670, Z    +0.000, E1   -25.472, E3 +458711.710}
SPL {X  -162.820, Y  +532.006, Z    +0.000, E1   -25.455, E3 +458722.167}
SPL {X  -162.820, Y  +534.806, Z    +0.000, E1   -25.465, E3 +458734.283}
SPL {X  -162.820, Y  +537.226, Z    +0.000, E1   -25.378, E3 +458745.565}
SPL {X  -162.820, Y  +540.345, Z    +0.000, E1   -25.451, E3 +458758.746}
SPL {X  -162.820, Y  +543.279, Z    +0.000, E1   -25.419, E3 +458771.779}
SPL {X  -162.820, Y  +546.125, Z    +0.000, E1   -25.505, E3 +458783.574}
SPL {X  -162.820, Y  +548.232, Z    +0.000, E1   -25.424, E3 +458793.336}
SPL {X  -162.820, Y  +550.399, Z    +0.000, E1   -25.424, E3 +458802.887}
SPL {X  -162.820, Y  +553.157, Z    +0.000, E1   -25.443, E3 +458814.861}
SPL {X  -162.820, Y  +556.150, Z    +0.000, E1   -25.445, E3 +458827.951}
SPL {X  -162.820, Y  +559.215, Z    +0.000, E1   -25.460, E3 +458841.252}
SPL {X  -162.820, Y  +562.125, Z    +0.000, E1   -25.434, E3 +458854.173}
SPL {X  -162.820, Y  +565.606, Z    +0.000, E1   -25.468, E3 +458869.302}
SPL {X  -162.820, Y  +568.974, Z    +0.000, E1   -25.453, E3 +458884.013}
SPL {X  -162.820, Y  +571.303, Z    +0.000, E1   -25.427, E3 +458894.359}
SPL {X  -162.820, Y  +574.067, Z    +0.000, E1   -25.459, E3 +458906.298}
SPL {X  -162.820, Y  +576.597, Z    +0.000, E1   -25.400, E3 +458917.770}
SPL {X  -162.820, Y  +578.977, Z    +0.000, E1   -25.460, E3 +458927.702}
SPL {X  -162.820, Y  +581.995, Z    +0.000, E1   -25.468, E3 +458941.060}
SPL {X  -162.820, Y  +585.512, Z    +0.000, E1   -25.448, E3 +458956.484}
SPL {X  -162.820, Y  +588.371, Z    +0.000, E1   -25.460, E3 +458968.870}
SPL {X  -162.820, Y  +590.476, Z    +0.000, E1   -25.398, E3 +458978.511}
SPL {X  -162.820, Y  +593.604, Z    +0.000, E1   -25.477, E3 +458991.789}
SPL {X  -162.820, Y  +596.868, Z    +0.000, E1   -25.461, E3 +459006.054}
SPL {X  -162.820, Y  +599.135, Z    +0.000, E1   -25.398, E3 +459016.423}
SPL {X  -162.820, Y  +601.296, Z    +0.000, E1   -25.399, E3 +459025.905}
SPL {X  -162.820, Y  +603.808, Z    +0.000, E1   -25.554, E3 +459035.693}
SPL {X  -162.820, Y  +607.007, Z    +0.000, E1   -25.491, E3 +459050.384}
SPL {X  -162.820, Y  +610.517, Z    +0.000, E1   -25.412, E3 +459066.176}
SPL {X  -162.820, Y  +613.762, Z    +0.000, E1   -25.472, E3 +459079.983}
SPL {X  -162.820, Y  +617.275, Z    +0.000, E1   -25.466, E3 +459095.422}
SPL {X  -162.820, Y  +621.264, Z    +0.000, E1   -25.514, E3 +459112.583}
SPL {X  -162.820, Y  +624.430, Z    +0.000, E1   -25.475, E3 +459126.514}
SPL {X  -162.820, Y  +626.570, Z    +0.000, E1   -25.441, E3 +459136.114}
SPL {X  -162.820, Y  +628.902, Z    +0.000, E1   -25.449, E3 +459146.294}
SPL {X  -162.820, Y  +631.177, Z    +0.000, E1   -25.467, E3 +459156.126}
SPL {X  -162.820, Y  +633.994, Z    +0.000, E1   -25.503, E3 +459168.172}
SPL {X  -162.820, Y  +637.619, Z    +0.000, E1   -25.497, E3 +459184.232}
SPL {X  -162.820, Y  +640.803, Z    +0.000, E1   -25.462, E3 +459198.195}
SPL {X  -162.820, Y  +643.028, Z    +0.000, E1   -25.494, E3 +459207.704}
SPL {X  -162.820, Y  +645.694, Z    +0.000, E1   -25.540, E3 +459218.992}
SPL {X  -162.820, Y  +649.102, Z    +0.000, E1   -25.495, E3 +459234.420}
SPL {X  -162.820, Y  +652.810, Z    +0.000, E1   -25.497, E3 +459250.453}
SPL {X  -162.820, Y  +655.214, Z    +0.000, E1   -25.485, E3 +459260.956}
SPL {X  -162.820, Y  +657.616, Z    +0.000, E1   -25.511, E3 +459271.310}
SPL {X  -162.820, Y  +660.851, Z    +0.000, E1   -25.520, E3 +459285.453}
SPL {X  -162.820, Y  +663.853, Z    +0.000, E1   -25.496, E3 +459298.635}
SPL {X  -162.820, Y  +666.096, Z    +0.000, E1   -25.408, E3 +459309.102}
SPL {X  -162.820, Y  +669.195, Z    +0.000, E1   -25.525, E3 +459321.939}
SPL {X  -162.820, Y  +672.979, Z    +0.000, E1   -25.478, E3 +459338.789}
SPL {X  -162.796, Y  +676.319, Z    +0.000, E1   -25.526, E3 +459352.934}
SPL {X  -162.739, Y  +678.625, Z    +0.000, E1   -25.423, E3 +459363.725}
SPL {X  -162.669, Y  +680.515, Z    +0.000, E1   -25.398, E3 +459372.179}
SPL {X  -162.545, Y  +682.952, Z    +0.000, E1   -25.510, E3 +459382.041}
SPL {X  -162.381, Y  +685.455, Z    +0.000, E1   -25.410, E3 +459393.728}
SPL {X  -162.102, Y  +688.774, Z    +0.000, E1   -25.417, E3 +459408.342}
SPL {X  -161.711, Y  +692.468, Z    +0.000, E1   -25.300, E3 +459425.315}
SPL {X  -161.141, Y  +696.825, Z    +0.000, E1   -26.170, E3 +459437.449}
SPL {X  -157.976, Y  +712.921, Z    +0.000, E1   -33.197, E3 +459447.990}
ENDSPLINE

SPLINE
SPL {X  -160.738, Y  +699.453, Z    +0.000, E1   -21.994, E3 +459485.617}
SPL {X  -161.689, Y  +692.657, Z    +0.000, E1   -15.656, E3 +459525.686}
SPL {X  -162.807, Y  +675.545, Z    +0.000, E1    -5.787, E3 +459521.186}
ENDSPLINE

SPLINE
SPL {X  -162.791, Y  +676.574, Z    +0.000, E1    -6.127, E3 +459534.289}
ENDSPLINE

SPLINE
SPL {X  -162.820, Y  +667.935, Z    +0.000, E1    -0.509, E3 +459524.375}
SPL {X  -162.820, Y  +662.949, Z    +0.000, E1    +3.113, E3 +459522.494}
SPL {X  -162.820, Y  +659.826, Z    +0.000, E1    +5.330, E3 +459529.598}
SPL {X  -162.820, Y  +656.907, Z    +0.000, E1    +7.703, E3 +459529.688}
SPL {X  -162.820, Y  +640.102, Z    +0.000, E1   +22.409, E3 +459524.378}
SPL {X  -162.820, Y  +633.503, Z    +0.000, E1   +21.975, E3 +459556.614}
SPL {X  -162.820, Y  +611.299, Z    +0.000, E1   +31.088, E3 +459584.727}
ENDSPLINE

SPLINE
SPL {X  -162.820, Y  +618.877, Z    +0.000, E1   +25.259, E3 +459596.221}
ENDSPLINE

SPLINE
SPL {X  -162.820, Y  +617.582, Z    +0.000, E1   +24.552, E3 +459607.598}
SPL {X  -162.820, Y  +614.716, Z    +0.000, E1   +24.535, E3 +459620.810}
SPL {X  -162.820, Y  +611.754, Z    +0.000, E1   +24.563, E3 +459634.098}
SPL {X  -162.820, Y  +608.970, Z    +0.000, E1   +24.542, E3 +459646.938}
SPL {X  -162.820, Y  +606.285, Z    +0.000, E1   +24.533, E3 +459659.273}
SPL {X  -162.820, Y  +603.509, Z    +0.000, E1   +24.546, E3 +459671.811}
SPL {X  -162.820, Y  +600.818, Z    +0.000, E1   +24.590, E3 +459683.733}
SPL {X  -162.820, Y  +598.053, Z    +0.000, E1   +24.547, E3 +459696.716}
SPL {X  -162.820, Y  +595.188, Z    +0.000, E1   +24.538, E3 +459709.805}
SPL {X  -162.820, Y  +592.738, Z    +0.000, E1   +24.551, E3 +459720.853}
SPL {X  -162.820, Y  +590.118, Z    +0.000, E1   +24.544, E3 +459732.912}
SPL {X  -162.820, Y  +587.204, Z    +0.000, E1   +24.592, E3 +459745.789}
SPL {X  -162.820, Y  +584.766, Z    +0.000, E1   +24.499, E3 +459757.622}
SPL {X  -162.820, Y  +581.896, Z    +0.000, E1   +24.528, E3 +459770.564}
SPL {X  -162.820, Y  +579.244, Z    +0.000, E1   +24.610, E3 +459781.909}
SPL {X  -162.820, Y  +576.848, Z    +0.000, E1   +24.543, E3 +459793.450}
SPL {X  -162.820, Y  +573.694, Z    +0.000, E1   +24.535, E3 +459807.919}
SPL {X  -162.820, Y  +571.322, Z    +0.000, E1   +24.492, E3 +459818.953}
SPL {X  -162.820, Y  +568.309, Z    +0.000, E1   +24.589, E3 +459832.178}
SPL {X  -162.820, Y  +564.977, Z    +0.000, E1   +24.571, E3 +459847.351}
SPL {X  -162.820, Y  +562.356, Z    +0.000, E1   +24.575, E3 +459859.250}
SPL {X  -162.820, Y  +560.119, Z    +0.000, E1   +24.506, E3 +459869.938}
SPL {X  -162.820, Y  +558.093, Z    +0.000, E1   +24.537, E3 +459878.956}
SPL {X  -162.820, Y  +555.584, Z    +0.000, E1   +24.559, E3 +459890.269}
SPL {X  -162.820, Y  +552.867, Z    +0.000, E1   +24.583, E3 +459902.464}
SPL {X  -162.820, Y  +549.589, Z    +0.000, E1   +24.547, E3 +459917.830}
SPL {X  -162.820, Y  +545.742, Z    +0.000, E1   +24.577, E3 +459935.117}
SPL {X  -162.820, Y  +542.970, Z    +0.000, E1   +24.579, E3 +459947.560}
SPL {X  -162.820, Y  +540.573, Z    +0.000, E1   +24.503, E3 +459959.194}
SPL {X  -162.820, Y  +538.106, Z    +0.000, E1   +24.553, E3 +459969.948}
SPL {X  -162.820, Y  +536.451, Z    +0.000, E1   +24.519, E3 +459977.766}
SPL {X  -162.820, Y  +534.025, Z    +0.000, E1   +24.589, E3 +459988.366}
SPL {X  -162.820, Y  +531.527, Z    +0.000, E1   +24.582, E3 +459999.752}
SPL {X  -162.820, Y  +529.165, Z    +0.000, E1   +24.521, E3 +460011.000}
SPL {X  -162.820, Y  +526.822, Z    +0.000, E1   +24.559, E3 +460021.364}
SPL {X  -162.820, Y  +524.112, Z    +0.000, E1   +24.542, E3 +460033.981}
SPL {X  -162.820, Y  +521.048, Z    +0.000, E1   +24.515, E3 +460048.118}
SPL {X  -162.820, Y  +518.185, Z    +0.000, E1   +24.561, E3 +460060.829}
SPL {X  -162.820, Y  +508.728, Z    +0.000, E1   +28.484, E3 +460071.368}
SPL {X  -162.820, Y  +500.664, Z    +0.000, E1   +31.476, E3 +460080.032}
SPL {X  -162.820, Y  +499.290, Z    +0.000, E1   +30.657, E3 +460090.315}
SPL {X  -162.820, Y  +497.251, Z    +0.000, E1   +29.634, E3 +460104.790}
SPL {X  -162.820, Y  +495.647, Z    +0.000, E1   +28.606, E3 +460117.666}
SPL {X  -162.820, Y  +494.678, Z    +0.000, E1   +27.647, E3 +460128.367}
SPL {X  -162.820, Y  +493.757, Z    +0.000, E1   +26.462, E3 +460140.727}
SPL {X  -162.820, Y  +491.420, Z    +0.000, E1   +25.780, E3 +460155.989}
SPL {X  -162.820, Y  +487.351, Z    +0.000, E1   +25.663, E3 +460174.505}
SPL {X  -162.820, Y  +484.247, Z    +0.000, E1   +25.651, E3 +460187.832}
SPL {X  -162.820, Y  +482.092, Z    +0.000, E1   +25.593, E3 +460197.659}
SPL {X  -162.820, Y  +479.578, Z    +0.000, E1   +25.634, E3 +460208.301}
SPL {X  -162.820, Y  +476.226, Z    +0.000, E1   +25.672, E3 +460222.692}
SPL {X  -162.820, Y  +473.037, Z    +0.000, E1   +25.618, E3 +460236.783}
SPL {X  -162.820, Y  +469.694, Z    +0.000, E1   +25.657, E3 +460251.157}
SPL {X  -162.820, Y  +465.727, Z    +0.000, E1   +25.676, E3 +460268.200}
SPL {X  -162.820, Y  +463.001, Z    +0.000, E1   +25.614, E3 +460280.317}
SPL {X  -162.820, Y  +459.882, Z    +0.000, E1   +25.674, E3 +460293.617}
SPL {X  -162.820, Y  +456.773, Z    +0.000, E1   +25.591, E3 +460307.563}
SPL {X  -162.820, Y  +454.429, Z    +0.000, E1   +25.642, E3 +460317.331}
SPL {X  -162.820, Y  +451.204, Z    +0.000, E1   +25.672, E3 +460331.358}
SPL {X  -162.820, Y  +447.822, Z    +0.000, E1   +25.664, E3 +460345.842}
SPL {X  -162.820, Y  +445.556, Z    +0.000, E1   +25.626, E3 +460355.972}
SPL {X  -162.820, Y  +443.328, Z    +0.000, E1   +25.642, E3 +460365.487}
SPL {X  -162.820, Y  +440.857, Z    +0.000, E1   +25.614, E3 +460376.521}
SPL {X  -162.820, Y  +437.636, Z    +0.000, E1   +25.597, E3 +460390.685}
SPL {X  -162.820, Y  +434.768, Z    +0.000, E1   +25.655, E3 +460402.586}
SPL {X  -162.820, Y  +431.823, Z    +0.000, E1   +25.651, E3 +460415.585}
SPL {X  -162.820, Y  +427.740, Z    +0.000, E1   +25.667, E3 +460433.213}
SPL {X  -162.820, Y  +423.655, Z    +0.000, E1   +25.628, E3 +460451.237}
SPL {X  -162.820, Y  +419.407, Z    +0.000, E1   +25.665, E3 +460469.430}
SPL {X  -162.820, Y  +415.900, Z    +0.000, E1   +25.638, E3 +460484.699}
SPL {X  -162.820, Y  +413.088, Z    +0.000, E1   +25.644, E3 +460496.855}
SPL {X  -162.820, Y  +410.320, Z    +0.000, E1   +25.604, E3 +460509.174}
SPL {X  -162.820, Y  +407.487, Z    +0.000, E1   +25.617, E3 +460521.382}
SPL {X  -162.820, Y  +404.293, Z    +0.000, E1   +25.628, E3 +460535.291}
SPL {X  -162.820, Y  +400.835, Z    +0.000, E1   +25.694, E3 +460549.691}
SPL {X  -162.820, Y  +398.703, Z    +0.000, E1   +25.586, E3 +460559.683}
SPL {X  -162.820, Y  +395.582, Z    +0.000, E1   +25.684, E3 +460572.675}
SPL {X  -162.820, Y  +391.417, Z    +0.000, E1   +25.659, E3 +460591.013}
SPL {X  -162.820, Y  +387.939, Z    +0.000, E1   +25.627, E3 +460606.159}
SPL {X  -162.820, Y  +385.565, Z    +0.000, E1   +25.686, E3 +460615.948}
SPL {X  -162.820, Y  +383.458, Z    +0.000, E1   +25.657, E3 +460625.312}
SPL {X  -162.820, Y  +380.448, Z    +0.000, E1   +25.674, E3 +460638.421}
SPL {X  -162.785, Y  +377.106, Z    +0.000, E1   +25.598, E3 +460653.365}
SPL {X  -162.709, Y  +374.484, Z    +0.000, E1   +25.711, E3 +460663.816}
SPL {X  -162.623, Y  +372.485, Z    +0.000, E1   +25.631, E3 +460673.097}
SPL {X  -162.487, Y  +370.088, Z    +0.000, E1   +25.525, E3 +460684.351}
SPL {X  -162.243, Y  +366.801, Z    +0.000, E1   +25.618, E3 +460697.991}
SPL {X  -161.977, Y  +363.953, Z    +0.000, E1   +25.528, E3 +460710.917}
SPL {X  -161.695, Y  +361.389, Z    +0.000, E1   +25.445, E3 +460722.733}
SPL {X  -161.190, Y  +357.520, Z    +0.000, E1   +25.774, E3 +460736.984}
SPL {X  -155.035, Y  +330.756, Z    +0.000, E1   +37.918, E3 +460747.485}
SPL {X  -153.918, Y  +327.401, Z    +0.000, E1   +34.677, E3 +460782.786}
ENDSPLINE

SPLINE
SPL {X  -159.701, Y  +348.785, Z    +0.000, E1   +24.361, E3 +460790.267}
SPL {X  -162.442, Y  +369.407, Z    +0.000, E1   +11.234, E3 +460819.902}
SPL {X  -162.820, Y  +384.333, Z    +0.000, E1    +1.902, E3 +460821.108}
SPL {X  -162.820, Y  +389.940, Z    +0.000, E1    -2.281, E3 +460824.029}
SPL {X  -162.820, Y  +396.652, Z    +0.000, E1    -7.520, E3 +460823.608}
SPL {X  -162.820, Y  +406.605, Z    +0.000, E1   -16.760, E3 +460816.085}
SPL {X  -162.820, Y  +420.013, Z    +0.000, E1   -22.833, E3 +460844.206}
SPL {X  -162.820, Y  +442.075, Z    +0.000, E1   -31.090, E3 +460876.992}
ENDSPLINE

SPLINE
SPL {X  -162.820, Y  +436.680, Z    +0.000, E1   -26.151, E3 +460890.296}
ENDSPLINE

SPLINE
SPL {X  -162.820, Y  +438.487, Z    +0.000, E1   -25.409, E3 +460903.935}
SPL {X  -162.820, Y  +441.593, Z    +0.000, E1   -25.391, E3 +460917.543}
SPL {X  -162.820, Y  +444.317, Z    +0.000, E1   -25.492, E3 +460928.724}
SPL {X  -162.820, Y  +447.641, Z    +0.000, E1   -25.460, E3 +460943.660}
SPL {X  -162.820, Y  +451.056, Z    +0.000, E1   -25.443, E3 +460958.603}
SPL {X  -162.820, Y  +454.662, Z    +0.000, E1   -25.474, E3 +460974.347}
SPL {X  -162.820, Y  +458.079, Z    +0.000, E1   -25.369, E3 +460989.926}
SPL {X  -162.820, Y  +460.719, Z    +0.000, E1   -25.411, E3 +461001.184}
SPL {X  -162.820, Y  +463.419, Z    +0.000, E1   -25.510, E3 +461012.222}
SPL {X  -162.820, Y  +465.376, Z    +0.000, E1   -25.372, E3 +461021.810}
SPL {X  -162.820, Y  +467.440, Z    +0.000, E1   -25.427, E3 +461030.441}
SPL {X  -162.820, Y  +470.010, Z    +0.000, E1   -25.445, E3 +461041.646}
SPL {X  -162.820, Y  +473.445, Z    +0.000, E1   -25.493, E3 +461056.370}
SPL {X  -162.820, Y  +476.157, Z    +0.000, E1   -25.426, E3 +461068.585}
SPL {X  -162.820, Y  +478.461, Z    +0.000, E1   -25.410, E3 +461078.865}
SPL {X  -162.820, Y  +481.644, Z    +0.000, E1   -25.433, E3 +461092.811}
SPL {X  -162.820, Y  +486.042, Z    +0.000, E1   -25.483, E3 +461111.730}
SPL {X  -162.820, Y  +490.287, Z    +0.000, E1   -25.463, E3 +461130.449}
SPL {X  -162.820, Y  +494.454, Z    +0.000, E1   -25.465, E3 +461148.680}
SPL {X  -162.820, Y  +498.644, Z    +0.000, E1   -25.463, E3 +461167.056}
SPL {X  -162.820, Y  +502.003, Z    +0.000, E1   -25.416, E3 +461181.954}
SPL {X  -162.820, Y  +505.370, Z    +0.000, E1   -25.456, E3 +461196.530}
SPL {X  -162.820, Y  +509.412, Z    +0.000, E1   -25.458, E3 +461214.253}
SPL {X  -162.820, Y  +512.406, Z    +0.000, E1   -25.425, E3 +461227.409}
SPL {X  -162.820, Y  +515.039, Z    +0.000, E1   -25.452, E3 +461238.819}
SPL {X  -162.820, Y  +518.350, Z    +0.000, E1   -25.425, E3 +461253.569}
SPL {X  -162.820, Y  +521.486, Z    +0.000, E1   -25.382, E3 +461267.597}
SPL {X  -162.820, Y  +524.180, Z    +0.000, E1   -25.495, E3 +461278.469}
SPL {X  -162.820, Y  +527.020, Z    +0.000, E1   -25.477, E3 +461291.162}
SPL {X  -162.820, Y  +529.670, Z    +0.000, E1   -25.472, E3 +461302.619}
SPL {X  -162.820, Y  +532.006, Z    +0.000, E1   -25.455, E3 +461313.076}
SPL {X  -162.820, Y  +534.806, Z    +0.000, E1   -25.465, E3 +461325.193}
SPL {X  -162.820, Y  +537.226, Z    +0.000, E1   -25.378, E3 +461336.474}
SPL {X  -162.820, Y  +540.345, Z    +0.000, E1   -25.451, E3 +461349.655}
SPL {X  -162.820, Y  +543.279, Z    +0.000, E1   -25.419, E3 +461362.688}
SPL {X  -162.820, Y  +546.125, Z    +0.000, E1   -25.505, E3 +461374.483}
SPL {X  -162.820, Y  +549.578, Z    +0.000, E1   -25.462, E3 +461390.107}
SPL {X  -162.820, Y  +553.157, Z    +0.000, E1   -25.443, E3 +461405.770}
SPL {X  -162.820, Y  +556.150, Z    +0.000, E1   -25.445, E3 +461418.860}
SPL {X  -162.820, Y  +559.215, Z    +0.000, E1   -25.460, E3 +461432.162}
SPL {X  -162.820, Y  +562.125, Z    +0.000, E1   -25.434, E3 +461445.082}
SPL {X  -162.820, Y  +564.880, Z    +0.000, E1   -25.448, E3 +461457.036}
SPL {X  -162.820, Y  +568.326, Z    +0.000, E1   -25.470, E3 +461472.095}
SPL {X  -162.820, Y  +571.303, Z    +0.000, E1   -25.427, E3 +461485.268}
SPL {X  -162.820, Y  +574.067, Z    +0.000, E1   -25.459, E3 +461497.207}
SPL {X  -162.820, Y  +576.597, Z    +0.000, E1   -25.400, E3 +461508.679}
SPL {X  -162.820, Y  +578.977, Z    +0.000, E1   -25.460, E3 +461518.611}
SPL {X  -162.820, Y  +581.995, Z    +0.000, E1   -25.468, E3 +461531.969}
SPL {X  -162.820, Y  +585.512, Z    +0.000, E1   -25.448, E3 +461547.393}
SPL {X  -162.820, Y  +588.371, Z    +0.000, E1   -25.460, E3 +461559.779}
SPL {X  -162.820, Y  +591.246, Z    +0.000, E1   -25.415, E3 +461572.798}
SPL {X  -162.820, Y  +594.339, Z    +0.000, E1   -25.487, E3 +461585.700}
SPL {X  -162.820, Y  +596.868, Z    +0.000, E1   -25.461, E3 +461596.964}
SPL {X  -162.820, Y  +600.326, Z    +0.000, E1   -25.438, E3 +461612.485}
SPL {X  -162.820, Y  +604.526, Z    +0.000, E1   -25.502, E3 +461630.308}
SPL {X  -162.820, Y  +607.811, Z    +0.000, E1   -25.507, E3 +461644.523}
SPL {X  -162.820, Y  +610.517, Z    +0.000, E1   -25.412, E3 +461657.085}
SPL {X  -162.820, Y  +613.762, Z    +0.000, E1   -25.472, E3 +461670.892}
SPL {X  -162.820, Y  +617.275, Z    +0.000, E1   -25.466, E3 +461686.331}
SPL {X  -162.820, Y  +621.264, Z    +0.000, E1   -25.514, E3 +461703.492}
SPL {X  -162.820, Y  +624.430, Z    +0.000, E1   -25.475, E3 +461717.423}
SPL {X  -162.820, Y  +626.570, Z    +0.000, E1   -25.441, E3 +461727.023}
SPL {X  -162.820, Y  +628.902, Z    +0.000, E1   -25.449, E3 +461737.203}
SPL {X  -162.820, Y  +631.177, Z    +0.000, E1   -25.467, E3 +461747.035}
SPL {X  -162.820, Y  +633.994, Z    +0.000, E1   -25.503, E3 +461759.081}
SPL {X  -162.820, Y  +636.469, Z    +0.000, E1   -25.465, E3 +461770.125}
SPL {X  -162.820, Y  +638.486, Z    +0.000, E1   -25.456, E3 +461779.042}
SPL {X  -162.820, Y  +640.803, Z    +0.000, E1   -25.462, E3 +461789.104}
SPL {X  -162.820, Y  +643.028, Z    +0.000, E1   -25.494, E3 +461798.613}
SPL {X  -162.820, Y  +645.694, Z    +0.000, E1   -25.540, E3 +461809.901}
SPL {X  -162.820, Y  +649.102, Z    +0.000, E1   -25.495, E3 +461825.329}
SPL {X  -162.820, Y  +652.810, Z    +0.000, E1   -25.497, E3 +461841.362}
SPL {X  -162.820, Y  +655.214, Z    +0.000, E1   -25.485, E3 +461851.865}
SPL {X  -162.820, Y  +657.616, Z    +0.000, E1   -25.511, E3 +461862.219}
SPL {X  -162.820, Y  +660.851, Z    +0.000, E1   -25.520, E3 +461876.362}
SPL {X  -162.820, Y  +663.853, Z    +0.000, E1   -25.496, E3 +461889.544}
SPL {X  -162.820, Y  +666.096, Z    +0.000, E1   -25.408, E3 +461900.011}
SPL {X  -162.820, Y  +669.195, Z    +0.000, E1   -25.525, E3 +461912.848}
SPL {X  -162.820, Y  +672.979, Z    +0.000, E1   -25.478, E3 +461929.698}
SPL {X  -162.796, Y  +676.319, Z    +0.000, E1   -25.526, E3 +461943.843}
SPL {X  -162.739, Y  +678.625, Z    +0.000, E1   -25.423, E3 +461954.634}
SPL {X  -162.669, Y  +680.515, Z    +0.000, E1   -25.398, E3 +461963.088}
SPL {X  -162.545, Y  +682.952, Z    +0.000, E1   -25.510, E3 +461972.950}
SPL {X  -162.381, Y  +685.455, Z    +0.000, E1   -25.410, E3 +461984.637}
SPL {X  -162.194, Y  +687.760, Z    +0.000, E1   -25.360, E3 +461995.073}
SPL {X  -161.866, Y  +691.104, Z    +0.000, E1   -25.383, E3 +462009.705}
SPL {X  -161.024, Y  +697.619, Z    +0.000, E1   -26.780, E3 +462026.935}
SPL {X  -157.189, Y  +715.948, Z    +0.000, E1   -34.218, E3 +462041.854}
ENDSPLINE

SPLINE
SPL {X  -157.848, Y  +713.428, Z    +0.000, E1   -28.857, E3 +462075.994}
SPL {X  -161.035, Y  +697.541, Z    +0.000, E1   -20.899, E3 +462076.513}
SPL {X  -161.689, Y  +692.657, Z    +0.000, E1   -15.656, E3 +462116.595}
SPL {X  -162.807, Y  +675.545, Z    +0.000, E1    -5.787, E3 +462112.095}
ENDSPLINE

SPLINE
SPL {X  -162.791, Y  +676.574, Z    +0.000, E1    -6.127, E3 +462125.198}
ENDSPLINE

SPLINE
SPL {X  -162.820, Y  +664.716, Z    +0.000, E1    +1.705, E3 +462114.072}
SPL {X  -162.820, Y  +658.484, Z    +0.000, E1    +6.336, E3 +462120.548}
SPL {X  -162.820, Y  +640.102, Z    +0.000, E1   +22.409, E3 +462115.287}
SPL {X  -162.820, Y  +633.503, Z    +0.000, E1   +21.975, E3 +462147.524}
SPL {X  -162.820, Y  +611.299, Z    +0.000, E1   +31.088, E3 +462175.636}
ENDSPLINE

SPLINE
SPL {X  -162.820, Y  +618.877, Z    +0.000, E1   +25.259, E3 +462187.130}
ENDSPLINE

SPLINE
SPL {X  -162.820, Y  +617.582, Z    +0.000, E1   +24.552, E3 +462198.507}
SPL {X  -162.820, Y  +614.716, Z    +0.000, E1   +24.535, E3 +462211.719}
SPL {X  -162.820, Y  +611.754, Z    +0.000, E1   +24.563, E3 +462225.007}
SPL {X  -162.820, Y  +608.970, Z    +0.000, E1   +24.542, E3 +462237.847}
SPL {X  -162.820, Y  +606.285, Z    +0.000, E1   +24.533, E3 +462250.182}
SPL {X  -162.820, Y  +603.509, Z    +0.000, E1   +24.546, E3 +462262.720}
SPL {X  -162.820, Y  +600.818, Z    +0.000, E1   +24.590, E3 +462274.643}
SPL {X  -162.820, Y  +598.053, Z    +0.000, E1   +24.547, E3 +462287.626}
SPL {X  -162.820, Y  +595.188, Z    +0.000, E1   +24.538, E3 +462300.714}
SPL {X  -162.820, Y  +592.738, Z    +0.000, E1   +24.551, E3 +462311.762}
SPL {X  -162.820, Y  +590.118, Z    +0.000, E1   +24.544, E3 +462323.821}
SPL {X  -162.820, Y  +587.204, Z    +0.000, E1   +24.592, E3 +462336.698}
SPL {X  -162.820, Y  +584.193, Z    +0.000, E1   +24.484, E3 +462351.408}
SPL {X  -162.820, Y  +580.163, Z    +0.000, E1   +24.634, E3 +462368.643}
SPL {X  -162.820, Y  +576.848, Z    +0.000, E1   +24.543, E3 +462384.359}
SPL {X  -162.820, Y  +574.433, Z    +0.000, E1   +24.551, E3 +462395.190}
SPL {X  -162.820, Y  +572.074, Z    +0.000, E1   +24.505, E3 +462406.461}
SPL {X  -162.820, Y  +569.438, Z    +0.000, E1   +24.562, E3 +462417.920}
SPL {X  -162.820, Y  +567.494, Z    +0.000, E1   +24.547, E3 +462426.930}
SPL {X  -162.820, Y  +564.977, Z    +0.000, E1   +24.571, E3 +462438.260}
SPL {X  -162.820, Y  +562.356, Z    +0.000, E1   +24.575, E3 +462450.159}
SPL {X  -162.820, Y  +560.119, Z    +0.000, E1   +24.506, E3 +462460.848}
SPL {X  -162.820, Y  +558.093, Z    +0.000, E1   +24.537, E3 +462469.865}
SPL {X  -162.820, Y  +555.584, Z    +0.000, E1   +24.559, E3 +462481.178}
SPL {X  -162.820, Y  +552.169, Z    +0.000, E1   +24.581, E3 +462496.747}
SPL {X  -162.820, Y  +548.932, Z    +0.000, E1   +24.540, E3 +462511.647}
SPL {X  -162.820, Y  +545.742, Z    +0.000, E1   +24.577, E3 +462526.026}
SPL {X  -162.820, Y  +542.142, Z    +0.000, E1   +24.582, E3 +462542.379}
SPL {X  -162.820, Y  +538.903, Z    +0.000, E1   +24.519, E3 +462557.595}
SPL {X  -162.820, Y  +536.451, Z    +0.000, E1   +24.519, E3 +462568.675}
SPL {X  -162.820, Y  +534.025, Z    +0.000, E1   +24.589, E3 +462579.275}
SPL {X  -162.820, Y  +531.527, Z    +0.000, E1   +24.582, E3 +462590.661}
SPL {X  -162.820, Y  +529.165, Z    +0.000, E1   +24.521, E3 +462601.910}
SPL {X  -162.820, Y  +526.822, Z    +0.000, E1   +24.559, E3 +462612.273}
SPL {X  -162.820, Y  +524.112, Z    +0.000, E1   +24.542, E3 +462624.890}
SPL {X  -162.820, Y  +521.048, Z    +0.000, E1   +24.515, E3 +462639.027}
SPL {X  -162.820, Y  +518.185, Z    +0.000, E1   +24.561, E3 +462651.738}
SPL {X  -162.820, Y  +508.728, Z    +0.000, E1   +28.484, E3 +462662.278}
SPL {X  -162.820, Y  +500.664, Z    +0.000, E1   +31.476, E3 +462670.942}
SPL {X  -162.820, Y  +499.290, Z    +0.000, E1   +30.657, E3 +462681.224}
SPL {X  -162.820, Y  +497.700, Z    +0.000, E1   +29.785, E3 +462692.838}
SPL {X  -162.820, Y  +495.915, Z    +0.000, E1   +28.861, E3 +462705.931}
SPL {X  -162.820, Y  +494.678, Z    +0.000, E1   +27.647, E3 +462719.276}
SPL {X  -162.820, Y  +493.757, Z    +0.000, E1   +26.462, E3 +462731.636}
SPL {X  -162.820, Y  +491.420, Z    +0.000, E1   +25.780, E3 +462746.898}
SPL {X  -162.820, Y  +487.351, Z    +0.000, E1   +25.663, E3 +462765.414}
SPL {X  -162.820, Y  +484.247, Z    +0.000, E1   +25.651, E3 +462778.741}
SPL {X  -162.820, Y  +482.092, Z    +0.000, E1   +25.593, E3 +462788.568}
SPL {X  -162.820, Y  +479.578, Z    +0.000, E1   +25.634, E3 +462799.210}
SPL {X  -162.820, Y  +477.137, Z    +0.000, E1   +25.632, E3 +462809.790}
SPL {X  -162.820, Y  +473.770, Z    +0.000, E1   +25.664, E3 +462824.335}
SPL {X  -162.820, Y  +469.694, Z    +0.000, E1   +25.657, E3 +462842.067}
SPL {X  -162.820, Y  +465.727, Z    +0.000, E1   +25.676, E3 +462859.110}
SPL {X  -162.820, Y  +463.001, Z    +0.000, E1   +25.614, E3 +462871.226}
SPL {X  -162.820, Y  +459.882, Z    +0.000, E1   +25.674, E3 +462884.526}
SPL {X  -162.820, Y  +456.773, Z    +0.000, E1   +25.591, E3 +462898.472}
SPL {X  -162.820, Y  +454.429, Z    +0.000, E1   +25.642, E3 +462908.240}
SPL {X  -162.820, Y  +451.204, Z    +0.000, E1   +25.672, E3 +462922.267}
SPL {X  -162.820, Y  +447.822, Z    +0.000, E1   +25.664, E3 +462936.751}
SPL {X  -162.820, Y  +445.556, Z    +0.000, E1   +25.626, E3 +462946.882}
SPL {X  -162.820, Y  +443.328, Z    +0.000, E1   +25.642, E3 +462956.396}
SPL {X  -162.820, Y  +440.857, Z    +0.000, E1   +25.614, E3 +462967.430}
SPL {X  -162.820, Y  +437.636, Z    +0.000, E1   +25.597, E3 +462981.594}
SPL {X  -162.820, Y  +434.768, Z    +0.000, E1   +25.655, E3 +462993.495}
SPL {X  -162.820, Y  +431.823, Z    +0.000, E1   +25.651, E3 +463006.494}
SPL {X  -162.820, Y  +427.740, Z    +0.000, E1   +25.667, E3 +463024.122}
SPL {X  -162.820, Y  +423.655, Z    +0.000, E1   +25.628, E3 +463042.147}
SPL {X  -162.820, Y  +419.407, Z    +0.000, E1   +25.665, E3 +463060.339}
SPL {X  -162.820, Y  +415.900, Z    +0.000, E1   +25.638, E3 +463075.608}
SPL {X  -162.820, Y  +413.088, Z    +0.000, E1   +25.644, E3 +463087.764}
SPL {X  -162.820, Y  +410.320, Z    +0.000, E1   +25.604, E3 +463100.083}
SPL {X  -162.820, Y  +407.487, Z    +0.000, E1   +25.617, E3 +463112.291}
SPL {X  -162.820, Y  +405.108, Z    +0.000, E1   +25.535, E3 +463123.259}
SPL {X  -162.820, Y  +401.373, Z    +0.000, E1   +25.736, E3 +463138.095}
SPL {X  -162.820, Y  +398.703, Z    +0.000, E1   +25.586, E3 +463150.592}
SPL {X  -162.820, Y  +395.582, Z    +0.000, E1   +25.684, E3 +463163.584}
SPL {X  -162.820, Y  +391.417, Z    +0.000, E1   +25.659, E3 +463181.922}
SPL {X  -162.820, Y  +387.939, Z    +0.000, E1   +25.627, E3 +463197.069}
SPL {X  -162.820, Y  +385.565, Z    +0.000, E1   +25.686, E3 +463206.857}
SPL {X  -162.820, Y  +383.458, Z    +0.000, E1   +25.657, E3 +463216.221}
SPL {X  -162.820, Y  +381.229, Z    +0.000, E1   +25.660, E3 +463225.897}
SPL {X  -162.797, Y  +377.786, Z    +0.000, E1   +25.638, E3 +463241.186}
SPL {X  -162.663, Y  +373.346, Z    +0.000, E1   +25.707, E3 +463259.925}
SPL {X  -162.487, Y  +370.088, Z    +0.000, E1   +25.525, E3 +463275.260}
SPL {X  -162.307, Y  +367.587, Z    +0.000, E1   +25.577, E3 +463285.678}
SPL {X  -162.041, Y  +364.588, Z    +0.000, E1   +25.591, E3 +463298.756}
SPL {X  -161.695, Y  +361.389, Z    +0.000, E1   +25.445, E3 +463313.642}
SPL {X  -161.364, Y  +358.774, Z    +0.000, E1   +25.454, E3 +463324.842}
SPL {X  -160.939, Y  +355.820, Z    +0.000, E1   +26.179, E3 +463332.060}
SPL {X  -155.035, Y  +330.756, Z    +0.000, E1   +37.918, E3 +463338.394}
SPL {X  -153.918, Y  +327.401, Z    +0.000, E1   +34.677, E3 +463373.695}
ENDSPLINE

SPLINE
SPL {X  -159.701, Y  +348.785, Z    +0.000, E1   +24.361, E3 +463381.176}
SPL {X  -162.442, Y  +369.407, Z    +0.000, E1   +11.234, E3 +463410.811}
SPL {X  -162.820, Y  +384.333, Z    +0.000, E1    +1.902, E3 +463412.017}
SPL {X  -162.820, Y  +389.940, Z    +0.000, E1    -2.281, E3 +463414.938}
SPL {X  -162.820, Y  +396.652, Z    +0.000, E1    -7.520, E3 +463414.517}
SPL {X  -162.820, Y  +409.181, Z    +0.000, E1   -18.650, E3 +463408.736}
SPL {X  -162.820, Y  +419.618, Z    +0.000, E1   -22.332, E3 +463436.218}
SPL {X  -162.820, Y  +442.075, Z    +0.000, E1   -31.090, E3 +463467.901}
ENDSPLINE

SPLINE
SPL {X  -162.820, Y  +436.949, Z    +0.000, E1   -25.871, E3 +463484.651}
ENDSPLINE

SPLINE
SPL {X  -162.820, Y  +439.120, Z    +0.000, E1   -25.352, E3 +463497.900}
SPL {X  -162.820, Y  +441.593, Z    +0.000, E1   -25.391, E3 +463508.452}
SPL {X  -162.820, Y  +444.317, Z    +0.000, E1   -25.492, E3 +463519.634}
SPL {X  -162.820, Y  +447.641, Z    +0.000, E1   -25.460, E3 +463534.569}
SPL {X  -162.820, Y  +451.939, Z    +0.000, E1   -25.468, E3 +463553.389}
SPL {X  -162.820, Y  +455.480, Z    +0.000, E1   -25.454, E3 +463568.800}
SPL {X  -162.820, Y  +458.079, Z    +0.000, E1   -25.369, E3 +463580.835}
SPL {X  -162.820, Y  +460.719, Z    +0.000, E1   -25.411, E3 +463592.094}
SPL {X  -162.820, Y  +463.419, Z    +0.000, E1   -25.510, E3 +463603.131}
SPL {X  -162.820, Y  +466.458, Z    +0.000, E1   -25.433, E3 +463617.187}
SPL {X  -162.820, Y  +470.010, Z    +0.000, E1   -25.445, E3 +463632.555}
SPL {X  -162.820, Y  +472.345, Z    +0.000, E1   -25.448, E3 +463642.642}
SPL {X  -162.820, Y  +475.191, Z    +0.000, E1   -25.489, E3 +463655.004}
SPL {X  -162.820, Y  +478.461, Z    +0.000, E1   -25.410, E3 +463669.774}
SPL {X  -162.820, Y  +480.780, Z    +0.000, E1   -25.447, E3 +463679.635}
SPL {X  -162.820, Y  +483.622, Z    +0.000, E1   -25.381, E3 +463692.677}
SPL {X  -162.820, Y  +486.874, Z    +0.000, E1   -25.478, E3 +463706.139}
SPL {X  -162.820, Y  +490.287, Z    +0.000, E1   -25.463, E3 +463721.358}
SPL {X  -162.820, Y  +494.454, Z    +0.000, E1   -25.465, E3 +463739.589}
SPL {X  -162.820, Y  +498.644, Z    +0.000, E1   -25.463, E3 +463757.965}
SPL {X  -162.820, Y  +502.845, Z    +0.000, E1   -25.458, E3 +463776.399}
SPL {X  -162.820, Y  +506.050, Z    +0.000, E1   -25.420, E3 +463790.538}
SPL {X  -162.820, Y  +508.346, Z    +0.000, E1   -25.444, E3 +463800.387}
SPL {X  -162.820, Y  +510.377, Z    +0.000, E1   -25.398, E3 +463809.632}
SPL {X  -162.820, Y  +513.176, Z    +0.000, E1   -25.443, E3 +463821.677}
SPL {X  -162.820, Y  +516.690, Z    +0.000, E1   -25.465, E3 +463836.888}
SPL {X  -162.820, Y  +519.134, Z    +0.000, E1   -25.366, E3 +463848.210}
SPL {X  -162.820, Y  +521.486, Z    +0.000, E1   -25.382, E3 +463858.506}
SPL {X  -162.820, Y  +524.180, Z    +0.000, E1   -25.495, E3 +463869.378}
SPL {X  -162.820, Y  +527.020, Z    +0.000, E1   -25.477, E3 +463882.071}
SPL {X  -162.820, Y  +529.670, Z    +0.000, E1   -25.472, E3 +463893.528}
SPL {X  -162.820, Y  +532.006, Z    +0.000, E1   -25.455, E3 +463903.985}
SPL {X  -162.820, Y  +534.806, Z    +0.000, E1   -25.465, E3 +463916.102}
SPL {X  -162.820, Y  +537.226, Z    +0.000, E1   -25.378, E3 +463927.383}
SPL {X  -162.820, Y  +540.345, Z    +0.000, E1   -25.451, E3 +463940.564}
SPL {X  -162.820, Y  +543.279, Z    +0.000, E1   -25.419, E3 +463953.597}
SPL {X  -162.820, Y  +546.125, Z    +0.000, E1   -25.505, E3 +463965.392}
SPL {X  -162.820, Y  +549.578, Z    +0.000, E1   -25.462, E3 +463981.016}
SPL {X  -162.820, Y  +553.157, Z    +0.000, E1   -25.443, E3 +463996.679}
SPL {X  -162.820, Y  +556.150, Z    +0.000, E1   -25.445, E3 +464009.769}
SPL {X  -162.820, Y  +559.215, Z    +0.000, E1   -25.460, E3 +464023.071}
SPL {X  -162.820, Y  +562.125, Z    +0.000, E1   -25.434, E3 +464035.991}
SPL {X  -162.820, Y  +564.880, Z    +0.000, E1   -25.448, E3 +464047.945}
SPL {X  -162.820, Y  +568.326, Z    +0.000, E1   -25.470, E3 +464063.005}
SPL {X  -162.820, Y  +571.303, Z    +0.000, E1   -25.427, E3 +464076.177}
SPL {X  -162.820, Y  +574.067, Z    +0.000, E1   -25.459, E3 +464088.116}
SPL {X  -162.820, Y  +576.597, Z    +0.000, E1   -25.400, E3 +464099.588}
SPL {X  -162.820, Y  +578.977, Z    +0.000, E1   -25.460, E3 +464109.520}
SPL {X  -162.820, Y  +581.995, Z    +0.000, E1   -25.468, E3 +464122.878}
SPL {X  -162.820, Y  +585.512, Z    +0.000, E1   -25.448, E3 +464138.302}
SPL {X  -162.820, Y  +588.371, Z    +0.000, E1   -25.460, E3 +464150.688}
SPL {X  -162.820, Y  +591.246, Z    +0.000, E1   -25.415, E3 +464163.707}
SPL {X  -162.820, Y  +594.339, Z    +0.000, E1   -25.487, E3 +464176.609}
SPL {X  -162.820, Y  +596.868, Z    +0.000, E1   -25.461, E3 +464187.873}
SPL {X  -162.820, Y  +600.326, Z    +0.000, E1   -25.438, E3 +464203.394}
SPL {X  -162.820, Y  +604.526, Z    +0.000, E1   -25.502, E3 +464221.217}
SPL {X  -162.820, Y  +607.811, Z    +0.000, E1   -25.507, E3 +464235.432}
SPL {X  -162.820, Y  +610.517, Z    +0.000, E1   -25.412, E3 +464247.994}
SPL {X  -162.820, Y  +613.762, Z    +0.000, E1   -25.472, E3 +464261.801}
SPL {X  -162.820, Y  +616.216, Z    +0.000, E1   -25.419, E3 +464272.797}
SPL {X  -162.820, Y  +618.995, Z    +0.000, E1   -25.483, E3 +464284.646}
SPL {X  -162.820, Y  +622.118, Z    +0.000, E1   -25.492, E3 +464298.111}
SPL {X  -162.820, Y  +624.430, Z    +0.000, E1   -25.475, E3 +464308.332}
SPL {X  -162.820, Y  +626.570, Z    +0.000, E1   -25.441, E3 +464317.932}
SPL {X  -162.820, Y  +628.902, Z    +0.000, E1   -25.449, E3 +464328.113}
SPL {X  -162.820, Y  +631.177, Z    +0.000, E1   -25.467, E3 +464337.944}
SPL {X  -162.820, Y  +633.994, Z    +0.000, E1   -25.503, E3 +464349.990}
SPL {X  -162.820, Y  +636.469, Z    +0.000, E1   -25.465, E3 +464361.034}
SPL {X  -162.820, Y  +638.486, Z    +0.000, E1   -25.456, E3 +464369.952}
SPL {X  -162.820, Y  +640.803, Z    +0.000, E1   -25.462, E3 +464380.013}
SPL {X  -162.820, Y  +643.028, Z    +0.000, E1   -25.494, E3 +464389.522}
SPL {X  -162.820, Y  +645.694, Z    +0.000, E1   -25.540, E3 +464400.810}
SPL {X  -162.820, Y  +649.102, Z    +0.000, E1   -25.495, E3 +464416.238}
SPL {X  -162.820, Y  +652.810, Z    +0.000, E1   -25.497, E3 +464432.272}
SPL {X  -162.820, Y  +655.214, Z    +0.000, E1   -25.485, E3 +464442.774}
SPL {X  -162.820, Y  +657.616, Z    +0.000, E1   -25.511, E3 +464453.129}
SPL {X  -162.820, Y  +660.007, Z    +0.000, E1   -25.550, E3 +464463.190}
SPL {X  -162.820, Y  +662.980, Z    +0.000, E1   -25.505, E3 +464476.748}
SPL {X  -162.820, Y  +667.253, Z    +0.000, E1   -25.483, E3 +464495.625}
SPL {X  -162.820, Y  +671.102, Z    +0.000, E1   -25.514, E3 +464512.076}
SPL {X  -162.820, Y  +673.648, Z    +0.000, E1   -25.431, E3 +464523.742}
SPL {X  -162.796, Y  +676.319, Z    +0.000, E1   -25.526, E3 +464534.752}
SPL {X  -162.739, Y  +678.625, Z    +0.000, E1   -25.423, E3 +464545.543}
SPL {X  -162.669, Y  +680.515, Z    +0.000, E1   -25.398, E3 +464553.997}
SPL {X  -162.545, Y  +682.952, Z    +0.000, E1   -25.510, E3 +464563.859}
SPL {X  -162.381, Y  +685.455, Z    +0.000, E1   -25.410, E3 +464575.546}
SPL {X  -162.102, Y  +688.774, Z    +0.000, E1   -25.417, E3 +464590.160}
SPL {X  -161.778, Y  +691.887, Z    +0.000, E1   -25.301, E3 +464604.462}
SPL {X  -161.319, Y  +695.558, Z    +0.000, E1   -25.832, E3 +464616.416}
SPL {X  -157.976, Y  +712.921, Z    +0.000, E1   -33.197, E3 +464629.808}
SPL {X  -157.848, Y  +713.428, Z    +0.000, E1   -28.857, E3 +464666.903}
ENDSPLINE

SPLINE
SPL {X  -161.035, Y  +697.541, Z    +0.000, E1   -20.899, E3 +464667.422}
ENDSPLINE

SPLINE
SPL {X  -160.945, Y  +698.140, Z    +0.000, E1   -18.412, E3 +464709.674}
ENDSPLINE

SPLINE
SPL {X  -162.497, Y  +683.755, Z    +0.000, E1   -10.754, E3 +464703.818}
SPL {X  -162.819, Y  +673.996, Z    +0.000, E1    -4.745, E3 +464703.419}
ENDSPLINE

SPLINE
SPL {X  -162.791, Y  +676.574, Z    +0.000, E1    -6.127, E3 +464716.107}
ENDSPLINE

SPLINE
SPL {X  -162.820, Y  +667.935, Z    +0.000, E1    -0.509, E3 +464706.193}
SPL {X  -162.820, Y  +662.949, Z    +0.000, E1    +3.113, E3 +464704.312}
SPL {X  -162.820, Y  +659.826, Z    +0.000, E1    +5.330, E3 +464711.416}
SPL {X  -162.820, Y  +656.907, Z    +0.000, E1    +7.703, E3 +464711.506}
SPL {X  -162.820, Y  +640.102, Z    +0.000, E1   +22.409, E3 +464706.196}
SPL {X  -162.820, Y  +633.503, Z    +0.000, E1   +21.975, E3 +464738.433}
SPL {X  -162.820, Y  +611.299, Z    +0.000, E1   +31.088, E3 +464766.545}
ENDSPLINE

SPLINE
SPL {X  -162.820, Y  +618.877, Z    +0.000, E1   +25.259, E3 +464778.040}
ENDSPLINE

SPLINE
SPL {X  -162.820, Y  +617.582, Z    +0.000, E1   +24.552, E3 +464789.416}
SPL {X  -162.820, Y  +614.716, Z    +0.000, E1   +24.535, E3 +464802.628}
SPL {X  -162.820, Y  +611.754, Z    +0.000, E1   +24.563, E3 +464815.916}
SPL {X  -162.820, Y  +608.970, Z    +0.000, E1   +24.542, E3 +464828.756}
SPL {X  -162.820, Y  +606.285, Z    +0.000, E1   +24.533, E3 +464841.092}
SPL {X  -162.820, Y  +603.509, Z    +0.000, E1   +24.546, E3 +464853.629}
SPL {X  -162.820, Y  +600.230, Z    +0.000, E1   +24.589, E3 +464868.374}
SPL {X  -162.820, Y  +597.446, Z    +0.000, E1   +24.542, E3 +464881.232}
SPL {X  -162.820, Y  +595.188, Z    +0.000, E1   +24.538, E3 +464891.623}
SPL {X  -162.820, Y  +592.738, Z    +0.000, E1   +24.551, E3 +464902.671}
SPL {X  -162.820, Y  +590.118, Z    +0.000, E1   +24.544, E3 +464914.731}
SPL {X  -162.820, Y  +587.204, Z    +0.000, E1   +24.592, E3 +464927.607}
SPL {X  -162.820, Y  +584.766, Z    +0.000, E1   +24.499, E3 +464939.441}
SPL {X  -162.820, Y  +581.896, Z    +0.000, E1   +24.528, E3 +464952.383}
SPL {X  -162.820, Y  +578.588, Z    +0.000, E1   +24.598, E3 +464966.934}
SPL {X  -162.820, Y  +576.196, Z    +0.000, E1   +24.519, E3 +464978.317}
SPL {X  -162.820, Y  +573.694, Z    +0.000, E1   +24.535, E3 +464989.738}
SPL {X  -162.820, Y  +570.310, Z    +0.000, E1   +24.556, E3 +465005.054}
SPL {X  -162.820, Y  +567.494, Z    +0.000, E1   +24.547, E3 +465017.839}
SPL {X  -162.820, Y  +564.977, Z    +0.000, E1   +24.571, E3 +465029.169}
SPL {X  -162.820, Y  +562.356, Z    +0.000, E1   +24.575, E3 +465041.068}
SPL {X  -162.820, Y  +558.990, Z    +0.000, E1   +24.558, E3 +465056.718}
SPL {X  -162.820, Y  +555.584, Z    +0.000, E1   +24.559, E3 +465072.087}
SPL {X  -162.820, Y  +552.867, Z    +0.000, E1   +24.583, E3 +465084.282}
SPL {X  -162.820, Y  +549.589, Z    +0.000, E1   +24.547, E3 +465099.648}
SPL {X  -162.820, Y  +545.742, Z    +0.000, E1   +24.577, E3 +465116.935}
SPL {X  -162.820, Y  +542.970, Z    +0.000, E1   +24.579, E3 +465129.378}
SPL {X  -162.820, Y  +540.573, Z    +0.000, E1   +24.503, E3 +465141.012}
SPL {X  -162.820, Y  +537.211, Z    +0.000, E1   +24.561, E3 +465155.941}
SPL {X  -162.820, Y  +534.025, Z    +0.000, E1   +24.589, E3 +465170.184}
SPL {X  -162.820, Y  +531.527, Z    +0.000, E1   +24.582, E3 +465181.570}
SPL {X  -162.820, Y  +529.165, Z    +0.000, E1   +24.521, E3 +465192.819}
SPL {X  -162.820, Y  +526.822, Z    +0.000, E1   +24.559, E3 +465203.182}
SPL {X  -162.820, Y  +524.112, Z    +0.000, E1   +24.542, E3 +465215.799}
SPL {X  -162.820, Y  +521.048, Z    +0.000, E1   +24.515, E3 +465229.936}
SPL {X  -162.820, Y  +518.185, Z    +0.000, E1   +24.561, E3 +465242.647}
SPL {X  -162.820, Y  +508.728, Z    +0.000, E1   +28.484, E3 +465253.187}
SPL {X  -162.820, Y  +500.664, Z    +0.000, E1   +31.476, E3 +465261.851}
SPL {X  -162.820, Y  +499.290, Z    +0.000, E1   +30.657, E3 +465272.133}
SPL {X  -162.820, Y  +497.251, Z    +0.000, E1   +29.634, E3 +465286.608}
SPL {X  -162.820, Y  +495.647, Z    +0.000, E1   +28.606, E3 +465299.485}
SPL {X  -162.820, Y  +494.678, Z    +0.000, E1   +27.647, E3 +465310.186}
SPL {X  -162.820, Y  +493.757, Z    +0.000, E1   +26.462, E3 +465322.546}
SPL {X  -162.820, Y  +492.330, Z    +0.000, E1   +25.953, E3 +465332.300}
SPL {X  -162.820, Y  +489.800, Z    +0.000, E1   +25.653, E3 +465345.761}
SPL {X  -162.820, Y  +485.392, Z    +0.000, E1   +25.667, E3 +465364.789}
SPL {X  -162.820, Y  +482.092, Z    +0.000, E1   +25.593, E3 +465379.477}
SPL {X  -162.820, Y  +479.578, Z    +0.000, E1   +25.634, E3 +465390.120}
SPL {X  -162.820, Y  +476.226, Z    +0.000, E1   +25.672, E3 +465404.510}
SPL {X  -162.820, Y  +473.037, Z    +0.000, E1   +25.618, E3 +465418.601}
SPL {X  -162.820, Y  +470.744, Z    +0.000, E1   +25.641, E3 +465428.341}
SPL {X  -162.820, Y  +467.745, Z    +0.000, E1   +25.668, E3 +465441.324}
SPL {X  -162.820, Y  +463.978, Z    +0.000, E1   +25.651, E3 +465457.801}
SPL {X  -162.820, Y  +459.882, Z    +0.000, E1   +25.674, E3 +465475.435}
SPL {X  -162.820, Y  +456.773, Z    +0.000, E1   +25.591, E3 +465489.382}
SPL {X  -162.820, Y  +454.429, Z    +0.000, E1   +25.642, E3 +465499.149}
SPL {X  -162.820, Y  +451.204, Z    +0.000, E1   +25.672, E3 +465513.176}
SPL {X  -162.820, Y  +447.822, Z    +0.000, E1   +25.664, E3 +465527.660}
SPL {X  -162.820, Y  +445.556, Z    +0.000, E1   +25.626, E3 +465537.791}
SPL {X  -162.820, Y  +443.328, Z    +0.000, E1   +25.642, E3 +465547.305}
SPL {X  -162.820, Y  +440.857, Z    +0.000, E1   +25.614, E3 +465558.339}
SPL {X  -162.820, Y  +437.636, Z    +0.000, E1   +25.597, E3 +465572.503}
SPL {X  -162.820, Y  +434.768, Z    +0.000, E1   +25.655, E3 +465584.404}
SPL {X  -162.820, Y  +431.823, Z    +0.000, E1   +25.651, E3 +465597.403}
SPL {X  -162.820, Y  +427.740, Z    +0.000, E1   +25.667, E3 +465615.031}
SPL {X  -162.820, Y  +423.655, Z    +0.000, E1   +25.628, E3 +465633.056}
SPL {X  -162.820, Y  +419.407, Z    +0.000, E1   +25.665, E3 +465651.248}
SPL {X  -162.820, Y  +415.900, Z    +0.000, E1   +25.638, E3 +465666.517}
SPL {X  -162.820, Y  +413.088, Z    +0.000, E1   +25.644, E3 +465678.674}
SPL {X  -162.820, Y  +410.320, Z    +0.000, E1   +25.604, E3 +465690.992}
SPL {X  -162.820, Y  +407.487, Z    +0.000, E1   +25.617, E3 +465703.200}
SPL {X  -162.820, Y  +405.108, Z    +0.000, E1   +25.535, E3 +465714.168}
SPL {X  -162.820, Y  +401.373, Z    +0.000, E1   +25.736, E3 +465729.004}
SPL {X  -162.820, Y  +397.357, Z    +0.000, E1   +25.652, E3 +465747.075}
SPL {X  -162.820, Y  +393.659, Z    +0.000, E1   +25.666, E3 +465762.875}
SPL {X  -162.820, Y  +390.679, Z    +0.000, E1   +25.624, E3 +465776.118}
SPL {X  -162.820, Y  +387.939, Z    +0.000, E1   +25.627, E3 +465787.978}
SPL {X  -162.820, Y  +384.398, Z    +0.000, E1   +25.707, E3 +465802.875}
SPL {X  -162.820, Y  +380.448, Z    +0.000, E1   +25.674, E3 +465820.239}
SPL {X  -162.785, Y  +377.106, Z    +0.000, E1   +25.598, E3 +465835.183}
SPL {X  -162.709, Y  +374.484, Z    +0.000, E1   +25.711, E3 +465845.634}
SPL {X  -162.623, Y  +372.485, Z    +0.000, E1   +25.631, E3 +465854.915}
SPL {X  -162.487, Y  +370.088, Z    +0.000, E1   +25.525, E3 +465866.169}
SPL {X  -162.243, Y  +366.801, Z    +0.000, E1   +25.618, E3 +465879.809}
SPL {X  -161.977, Y  +363.953, Z    +0.000, E1   +25.528, E3 +465892.736}
SPL {X  -161.695, Y  +361.389, Z    +0.000, E1   +25.445, E3 +465904.551}
SPL {X  -161.364, Y  +358.774, Z    +0.000, E1   +25.454, E3 +465915.751}
SPL {X  -160.939, Y  +355.820, Z    +0.000, E1   +26.179, E3 +465922.969}
SPL {X  -155.035, Y  +330.756, Z    +0.000, E1   +37.918, E3 +465929.303}
SPL {X  -153.918, Y  +327.401, Z    +0.000, E1   +34.677, E3 +465964.604}
ENDSPLINE

SPLINE
SPL {X  -159.701, Y  +348.785, Z    +0.000, E1   +24.361, E3 +465972.085}
SPL {X  -162.442, Y  +369.407, Z    +0.000, E1   +11.234, E3 +466001.720}
SPL {X  -162.820, Y  +384.333, Z    +0.000, E1    +1.902, E3 +466002.926}
SPL {X  -162.820, Y  +389.940, Z    +0.000, E1    -2.281, E3 +466005.847}
SPL {X  -162.820, Y  +396.652, Z    +0.000, E1    -7.520, E3 +466005.426}
SPL {X  -162.820, Y  +406.605, Z    +0.000, E1   -16.760, E3 +465997.903}
SPL {X  -162.820, Y  +418.675, Z    +0.000, E1   -22.201, E3 +466024.151}
SPL {X  -162.820, Y  +425.113, Z    +0.000, E1   -25.243, E3 +466033.088}
SPL {X  -162.820, Y  +441.937, Z    +0.000, E1   -31.578, E3 +466055.166}
ENDSPLINE

SPLINE
SPL {X  -162.820, Y  +437.771, Z    +0.000, E1   -26.555, E3 +466074.266}
ENDSPLINE

SPLINE
SPL {X  -162.820, Y  +439.120, Z    +0.000, E1   -25.352, E3 +466088.809}
SPL {X  -162.820, Y  +441.593, Z    +0.000, E1   -25.391, E3 +466099.361}
SPL {X  -162.820, Y  +444.317, Z    +0.000, E1   -25.492, E3 +466110.543}
SPL {X  -162.820, Y  +446.544, Z    +0.000, E1   -25.427, E3 +466120.712}
SPL {X  -162.820, Y  +448.500, Z    +0.000, E1   -25.425, E3 +466129.314}
SPL {X  -162.820, Y  +451.056, Z    +0.000, E1   -25.443, E3 +466140.421}
SPL {X  -162.820, Y  +454.662, Z    +0.000, E1   -25.474, E3 +466156.165}
SPL {X  -162.820, Y  +458.079, Z    +0.000, E1   -25.369, E3 +466171.745}
SPL {X  -162.820, Y  +460.719, Z    +0.000, E1   -25.411, E3 +466183.003}
SPL {X  -162.820, Y  +463.419, Z    +0.000, E1   -25.510, E3 +466194.040}
SPL {X  -162.820, Y  +465.376, Z    +0.000, E1   -25.372, E3 +466203.628}
SPL {X  -162.820, Y  +467.440, Z    +0.000, E1   -25.427, E3 +466212.260}
SPL {X  -162.820, Y  +470.010, Z    +0.000, E1   -25.445, E3 +466223.464}
SPL {X  -162.820, Y  +473.445, Z    +0.000, E1   -25.493, E3 +466238.188}
SPL {X  -162.820, Y  +476.157, Z    +0.000, E1   -25.426, E3 +466250.403}
SPL {X  -162.820, Y  +478.461, Z    +0.000, E1   -25.410, E3 +466260.683}
SPL {X  -162.820, Y  +481.644, Z    +0.000, E1   -25.433, E3 +466274.629}
SPL {X  -162.820, Y  +486.042, Z    +0.000, E1   -25.483, E3 +466293.548}
SPL {X  -162.820, Y  +490.287, Z    +0.000, E1   -25.463, E3 +466312.267}
SPL {X  -162.820, Y  +494.454, Z    +0.000, E1   -25.465, E3 +466330.498}
SPL {X  -162.820, Y  +498.644, Z    +0.000, E1   -25.463, E3 +466348.874}
SPL {X  -162.820, Y  +502.845, Z    +0.000, E1   -25.458, E3 +466367.308}
SPL {X  -162.820, Y  +506.050, Z    +0.000, E1   -25.420, E3 +466381.447}
SPL {X  -162.820, Y  +508.346, Z    +0.000, E1   -25.444, E3 +466391.296}
SPL {X  -162.820, Y  +510.377, Z    +0.000, E1   -25.398, E3 +466400.541}
SPL {X  -162.820, Y  +513.176, Z    +0.000, E1   -25.443, E3 +466412.586}
SPL {X  -162.820, Y  +516.690, Z    +0.000, E1   -25.465, E3 +466427.797}
SPL {X  -162.820, Y  +519.134, Z    +0.000, E1   -25.366, E3 +466439.119}
SPL {X  -162.820, Y  +521.486, Z    +0.000, E1   -25.382, E3 +466449.415}
SPL {X  -162.820, Y  +524.180, Z    +0.000, E1   -25.495, E3 +466460.287}
SPL {X  -162.820, Y  +527.020, Z    +0.000, E1   -25.477, E3 +466472.980}
SPL {X  -162.820, Y  +529.670, Z    +0.000, E1   -25.472, E3 +466484.437}
SPL {X  -162.820, Y  +532.006, Z    +0.000, E1   -25.455, E3 +466494.894}
SPL {X  -162.820, Y  +534.806, Z    +0.000, E1   -25.465, E3 +466507.011}
SPL {X  -162.820, Y  +537.226, Z    +0.000, E1   -25.378, E3 +466518.292}
SPL {X  -162.820, Y  +540.345, Z    +0.000, E1   -25.451, E3 +466531.473}
SPL {X  -162.820, Y  +543.279, Z    +0.000, E1   -25.419, E3 +466544.506}
SPL {X  -162.820, Y  +546.125, Z    +0.000, E1   -25.505, E3 +466556.301}
SPL {X  -162.820, Y  +549.578, Z    +0.000, E1   -25.462, E3 +466571.925}
SPL {X  -162.820, Y  +553.157, Z    +0.000, E1   -25.443, E3 +466587.588}
SPL {X  -162.820, Y  +556.150, Z    +0.000, E1   -25.445, E3 +466600.678}
SPL {X  -162.820, Y  +559.215, Z    +0.000, E1   -25.460, E3 +466613.980}
SPL {X  -162.820, Y  +562.125, Z    +0.000, E1   -25.434, E3 +466626.900}
SPL {X  -162.820, Y  +564.880, Z    +0.000, E1   -25.448, E3 +466638.854}
SPL {X  -162.820, Y  +568.326, Z    +0.000, E1   -25.470, E3 +466653.914}
SPL {X  -162.820, Y  +571.303, Z    +0.000, E1   -25.427, E3 +466667.086}
SPL {X  -162.820, Y  +574.067, Z    +0.000, E1   -25.459, E3 +466679.025}
SPL {X  -162.820, Y  +576.597, Z    +0.000, E1   -25.400, E3 +466690.497}
SPL {X  -162.820, Y  +578.977, Z    +0.000, E1   -25.460, E3 +466700.429}
SPL {X  -162.820, Y  +581.995, Z    +0.000, E1   -25.468, E3 +466713.787}
SPL {X  -162.820, Y  +585.512, Z    +0.000, E1   -25.448, E3 +466729.211}
SPL {X  -162.820, Y  +588.371, Z    +0.000, E1   -25.460, E3 +466741.597}
SPL {X  -162.820, Y  +591.246, Z    +0.000, E1   -25.415, E3 +466754.616}
SPL {X  -162.820, Y  +594.339, Z    +0.000, E1   -25.487, E3 +466767.519}
SPL {X  -162.820, Y  +596.868, Z    +0.000, E1   -25.461, E3 +466778.782}
SPL {X  -162.820, Y  +599.135, Z    +0.000, E1   -25.398, E3 +466789.151}
SPL {X  -162.820, Y  +601.296, Z    +0.000, E1   -25.399, E3 +466798.632}
SPL {X  -162.820, Y  +603.808, Z    +0.000, E1   -25.554, E3 +466808.420}
SPL {X  -162.820, Y  +607.007, Z    +0.000, E1   -25.491, E3 +466823.111}
SPL {X  -162.820, Y  +611.438, Z    +0.000, E1   -25.467, E3 +466842.701}
SPL {X  -162.820, Y  +615.388, Z    +0.000, E1   -25.455, E3 +466859.960}
SPL {X  -162.820, Y  +618.103, Z    +0.000, E1   -25.456, E3 +466871.708}
SPL {X  -162.820, Y  +621.264, Z    +0.000, E1   -25.514, E3 +466885.310}
SPL {X  -162.820, Y  +624.430, Z    +0.000, E1   -25.475, E3 +466899.241}
SPL {X  -162.820, Y  +626.570, Z    +0.000, E1   -25.441, E3 +466908.842}
SPL {X  -162.820, Y  +628.902, Z    +0.000, E1   -25.449, E3 +466919.022}
SPL {X  -162.820, Y  +631.177, Z    +0.000, E1   -25.467, E3 +466928.853}
SPL {X  -162.820, Y  +633.994, Z    +0.000, E1   -25.503, E3 +466940.899}
SPL {X  -162.820, Y  +636.469, Z    +0.000, E1   -25.465, E3 +466951.943}
SPL {X  -162.820, Y  +638.486, Z    +0.000, E1   -25.456, E3 +466960.861}
SPL {X  -162.820, Y  +640.803, Z    +0.000, E1   -25.462, E3 +466970.922}
SPL {X  -162.820, Y  +643.028, Z    +0.000, E1   -25.494, E3 +466980.432}
SPL {X  -162.820, Y  +645.694, Z    +0.000, E1   -25.540, E3 +466991.719}
SPL {X  -162.820, Y  +649.102, Z    +0.000, E1   -25.495, E3 +467007.147}
SPL {X  -162.820, Y  +652.810, Z    +0.000, E1   -25.497, E3 +467023.181}
SPL {X  -162.820, Y  +655.214, Z    +0.000, E1   -25.485, E3 +467033.683}
SPL {X  -162.820, Y  +657.616, Z    +0.000, E1   -25.511, E3 +467044.038}
SPL {X  -162.820, Y  +660.007, Z    +0.000, E1   -25.550, E3 +467054.099}
SPL {X  -162.820, Y  +662.980, Z    +0.000, E1   -25.505, E3 +467067.657}
SPL {X  -162.820, Y  +667.253, Z    +0.000, E1   -25.483, E3 +467086.534}
SPL {X  -162.820, Y  +671.102, Z    +0.000, E1   -25.514, E3 +467102.985}
SPL {X  -162.820, Y  +673.648, Z    +0.000, E1   -25.431, E3 +467114.651}
SPL {X  -162.796, Y  +676.319, Z    +0.000, E1   -25.526, E3 +467125.661}
SPL {X  -162.739, Y  +678.625, Z    +0.000, E1   -25.423, E3 +467136.452}
SPL {X  -162.669, Y  +680.515, Z    +0.000, E1   -25.398, E3 +467144.907}
SPL {X  -162.545, Y  +682.952, Z    +0.000, E1   -25.510, E3 +467154.768}
SPL {X  -162.381, Y  +685.455, Z    +0.000, E1   -25.410, E3 +467166.455}
SPL {X  -162.194, Y  +687.760, Z    +0.000, E1   -25.360, E3 +467176.891}
SPL {X  -161.987, Y  +689.945, Z    +0.000, E1   -25.406, E3 +467186.043}
SPL {X  -161.711, Y  +692.468, Z    +0.000, E1   -25.300, E3 +467198.042}
SPL {X  -161.141, Y  +696.825, Z    +0.000, E1   -26.170, E3 +467210.176}
SPL {X  -157.976, Y  +712.921, Z    +0.000, E1   -33.197, E3 +467220.717}
ENDSPLINE

SPLINE
SPL {X  -160.738, Y  +699.453, Z    +0.000, E1   -21.994, E3 +467258.344}
SPL {X  -160.945, Y  +698.140, Z    +0.000, E1   -18.412, E3 +467300.584}
SPL {X  -162.497, Y  +683.755, Z    +0.000, E1   -10.754, E3 +467294.727}
SPL {X  -162.819, Y  +673.996, Z    +0.000, E1    -4.745, E3 +467294.328}
ENDSPLINE

SPLINE
SPL {X  -162.791, Y  +676.574, Z    +0.000, E1    -6.127, E3 +467307.016}
ENDSPLINE

SPLINE
SPL {X  -162.820, Y  +667.935, Z    +0.000, E1    -0.509, E3 +467297.102}
SPL {X  -162.820, Y  +662.949, Z    +0.000, E1    +3.113, E3 +467295.221}
SPL {X  -162.820, Y  +658.484, Z    +0.000, E1    +6.336, E3 +467302.367}
SPL {X  -162.820, Y  +640.102, Z    +0.000, E1   +22.409, E3 +467297.105}
SPL {X  -162.820, Y  +633.503, Z    +0.000, E1   +21.975, E3 +467329.342}
SPL {X  -162.820, Y  +611.299, Z    +0.000, E1   +31.088, E3 +467357.454}
ENDSPLINE

SPLINE
SPL {X  -162.820, Y  +618.877, Z    +0.000, E1   +25.259, E3 +467368.949}
ENDSPLINE

SPLINE
SPL {X  -162.820, Y  +617.582, Z    +0.000, E1   +24.552, E3 +467380.325}
SPL {X  -162.820, Y  +614.716, Z    +0.000, E1   +24.535, E3 +467393.537}
SPL {X  -162.820, Y  +611.754, Z    +0.000, E1   +24.563, E3 +467406.825}
SPL {X  -162.820, Y  +608.970, Z    +0.000, E1   +24.542, E3 +467419.665}
SPL {X  -162.820, Y  +606.285, Z    +0.000, E1   +24.533, E3 +467432.001}
SPL {X  -162.820, Y  +603.509, Z    +0.000, E1   +24.546, E3 +467444.538}
SPL {X  -162.820, Y  +600.818, Z    +0.000, E1   +24.590, E3 +467456.461}
SPL {X  -162.820, Y  +598.053, Z    +0.000, E1   +24.547, E3 +467469.444}
SPL {X  -162.820, Y  +595.188, Z    +0.000, E1   +24.538, E3 +467482.532}
SPL {X  -162.820, Y  +592.738, Z    +0.000, E1   +24.551, E3 +467493.580}
SPL {X  -162.820, Y  +590.118, Z    +0.000, E1   +24.544, E3 +467505.640}
SPL {X  -162.820, Y  +587.204, Z    +0.000, E1   +24.592, E3 +467518.517}
SPL {X  -162.820, Y  +584.766, Z    +0.000, E1   +24.499, E3 +467530.350}
SPL {X  -162.820, Y  +581.896, Z    +0.000, E1   +24.528, E3 +467543.292}
SPL {X  -162.820, Y  +578.588, Z    +0.000, E1   +24.598, E3 +467557.843}
SPL {X  -162.820, Y  +576.196, Z    +0.000, E1   +24.519, E3 +467569.227}
SPL {X  -162.820, Y  +573.694, Z    +0.000, E1   +24.535, E3 +467580.647}
SPL {X  -162.820, Y  +570.310, Z    +0.000, E1   +24.556, E3 +467595.963}
SPL {X  -162.820, Y  +567.494, Z    +0.000, E1   +24.547, E3 +467608.748}
SPL {X  -162.820, Y  +564.977, Z    +0.000, E1   +24.571, E3 +467620.078}
SPL {X  -162.820, Y  +562.356, Z    +0.000, E1   +24.575, E3 +467631.977}
SPL {X  -162.820, Y  +558.990, Z    +0.000, E1   +24.558, E3 +467647.627}
SPL {X  -162.820, Y  +555.584, Z    +0.000, E1   +24.559, E3 +467662.996}
SPL {X  -162.820, Y  +552.867, Z    +0.000, E1   +24.583, E3 +467675.191}
SPL {X  -162.820, Y  +549.589, Z    +0.000, E1   +24.547, E3 +467690.557}
SPL {X  -162.820, Y  +545.742, Z    +0.000, E1   +24.577, E3 +467707.844}
SPL {X  -162.820, Y  +542.970, Z    +0.000, E1   +24.579, E3 +467720.287}
SPL {X  -162.820, Y  +540.573, Z    +0.000, E1   +24.503, E3 +467731.921}
SPL {X  -162.820, Y  +537.211, Z    +0.000, E1   +24.561, E3 +467746.850}
SPL {X  -162.820, Y  +534.025, Z    +0.000, E1   +24.589, E3 +467761.093}
SPL {X  -162.820, Y  +531.527, Z    +0.000, E1   +24.582, E3 +467772.479}
SPL {X  -162.820, Y  +529.165, Z    +0.000, E1   +24.521, E3 +467783.728}
SPL {X  -162.820, Y  +526.822, Z    +0.000, E1   +24.559, E3 +467794.091}
SPL {X  -162.820, Y  +524.112, Z    +0.000, E1   +24.542, E3 +467806.708}
SPL {X  -162.820, Y  +521.048, Z    +0.000, E1   +24.515, E3 +467820.845}
SPL {X  -162.820, Y  +518.185, Z    +0.000, E1   +24.561, E3 +467833.556}
SPL {X  -162.820, Y  +508.728, Z    +0.000, E1   +28.484, E3 +467844.096}
SPL {X  -162.820, Y  +500.664, Z    +0.000, E1   +31.476, E3 +467852.760}
SPL {X  -162.820, Y  +499.290, Z    +0.000, E1   +30.657, E3 +467863.042}
SPL {X  -162.820, Y  +497.251, Z    +0.000, E1   +29.634, E3 +467877.518}
SPL {X  -162.820, Y  +495.647, Z    +0.000, E1   +28.606, E3 +467890.394}
SPL {X  -162.820, Y  +494.678, Z    +0.000, E1   +27.647, E3 +467901.095}
SPL {X  -162.820, Y  +493.757, Z    +0.000, E1   +26.462, E3 +467913.455}
SPL {X  -162.820, Y  +492.330, Z    +0.000, E1   +25.953, E3 +467923.209}
SPL {X  -162.820, Y  +489.800, Z    +0.000, E1   +25.653, E3 +467936.670}
SPL {X  -162.820, Y  +485.392, Z    +0.000, E1   +25.667, E3 +467955.698}
SPL {X  -162.820, Y  +482.092, Z    +0.000, E1   +25.593, E3 +467970.386}
SPL {X  -162.820, Y  +479.578, Z    +0.000, E1   +25.634, E3 +467981.029}
SPL {X  -162.820, Y  +476.226, Z    +0.000, E1   +25.672, E3 +467995.419}
SPL {X  -162.820, Y  +473.037, Z    +0.000, E1   +25.618, E3 +468009.510}
SPL {X  -162.820, Y  +470.744, Z    +0.000, E1   +25.641, E3 +468019.251}
SPL {X  -162.820, Y  +468.774, Z    +0.000, E1   +25.605, E3 +468028.079}
SPL {X  -162.820, Y  +465.727, Z    +0.000, E1   +25.676, E3 +468040.928}
SPL {X  -162.820, Y  +461.675, Z    +0.000, E1   +25.655, E3 +468058.734}
SPL {X  -162.820, Y  +457.479, Z    +0.000, E1   +25.656, E3 +468076.914}
SPL {X  -162.820, Y  +453.678, Z    +0.000, E1   +25.652, E3 +468093.366}
SPL {X  -162.820, Y  +450.466, Z    +0.000, E1   +25.644, E3 +468107.311}
SPL {X  -162.820, Y  +447.822, Z    +0.000, E1   +25.664, E3 +468118.569}
SPL {X  -162.820, Y  +444.499, Z    +0.000, E1   +25.673, E3 +468133.139}
SPL {X  -162.820, Y  +440.857, Z    +0.000, E1   +25.614, E3 +468149.248}
SPL {X  -162.820, Y  +438.582, Z    +0.000, E1   +25.544, E3 +468159.568}
SPL {X  -162.820, Y  +435.635, Z    +0.000, E1   +25.661, E3 +468171.663}
SPL {X  -162.820, Y  +432.815, Z    +0.000, E1   +25.641, E3 +468183.892}
SPL {X  -162.820, Y  +430.942, Z    +0.000, E1   +25.597, E3 +468192.360}
SPL {X  -162.820, Y  +428.576, Z    +0.000, E1   +25.647, E3 +468202.298}
SPL {X  -162.820, Y  +425.120, Z    +0.000, E1   +25.647, E3 +468217.482}
SPL {X  -162.820, Y  +420.840, Z    +0.000, E1   +25.658, E3 +468235.988}
SPL {X  -162.820, Y  +416.590, Z    +0.000, E1   +25.659, E3 +468254.433}
SPL {X  -162.820, Y  +412.302, Z    +0.000, E1   +25.662, E3 +468273.038}
SPL {X  -162.820, Y  +408.133, Z    +0.000, E1   +25.637, E3 +468291.296}
SPL {X  -162.820, Y  +404.293, Z    +0.000, E1   +25.628, E3 +468308.019}
SPL {X  -162.820, Y  +400.835, Z    +0.000, E1   +25.694, E3 +468322.418}
SPL {X  -162.820, Y  +398.703, Z    +0.000, E1   +25.586, E3 +468332.410}
SPL {X  -162.820, Y  +395.582, Z    +0.000, E1   +25.684, E3 +468345.402}
SPL {X  -162.820, Y  +391.417, Z    +0.000, E1   +25.659, E3 +468363.740}
SPL {X  -162.820, Y  +387.939, Z    +0.000, E1   +25.627, E3 +468378.887}
SPL {X  -162.820, Y  +385.565, Z    +0.000, E1   +25.686, E3 +468388.676}
SPL {X  -162.820, Y  +383.458, Z    +0.000, E1   +25.657, E3 +468398.040}
SPL {X  -162.820, Y  +381.229, Z    +0.000, E1   +25.660, E3 +468407.715}
SPL {X  -162.797, Y  +377.786, Z    +0.000, E1   +25.638, E3 +468423.004}
SPL {X  -162.663, Y  +373.346, Z    +0.000, E1   +25.707, E3 +468441.743}
SPL {X  -162.487, Y  +370.088, Z    +0.000, E1   +25.525, E3 +468457.078}
SPL {X  -162.243, Y  +366.801, Z    +0.000, E1   +25.618, E3 +468470.718}
SPL {X  -161.882, Y  +363.046, Z    +0.000, E1   +25.550, E3 +468487.602}
SPL {X  -161.454, Y  +359.455, Z    +0.000, E1   +25.428, E3 +468503.996}
SPL {X  -160.939, Y  +355.820, Z    +0.000, E1   +26.179, E3 +468513.879}
SPL {X  -154.424, Y  +328.890, Z    +0.000, E1   +36.591, E3 +468534.711}
ENDSPLINE

SPLINE
SPL {X  -159.701, Y  +348.785, Z    +0.000, E1   +24.361, E3 +468562.994}
SPL {X  -161.904, Y  +363.251, Z    +0.000, E1   +14.606, E3 +468592.789}
SPL {X  -162.745, Y  +375.561, Z    +0.000, E1    +7.538, E3 +468592.986}
SPL {X  -162.820, Y  +385.424, Z    +0.000, E1    +1.080, E3 +468593.880}
SPL {X  -162.820, Y  +389.940, Z    +0.000, E1    -2.281, E3 +468596.756}
SPL {X  -162.820, Y  +396.652, Z    +0.000, E1    -7.520, E3 +468596.335}
SPL {X  -162.820, Y  +406.605, Z    +0.000, E1   -16.760, E3 +468588.812}
SPL {X  -162.820, Y  +420.013, Z    +0.000, E1   -22.833, E3 +468616.933}
SPL {X  -162.820, Y  +442.075, Z    +0.000, E1   -31.090, E3 +468649.719}
ENDSPLINE

SPLINE
SPL {X  -162.820, Y  +436.680, Z    +0.000, E1   -26.151, E3 +468663.023}
ENDSPLINE

